(* IEC 61131-3 sources: uPC2_EMCTEST/UPC2_EMCTEST/UPC2_EMCTEST/Source/Programs, 11 files *)

(* ---- HeosTestMain.st ---- *)
USING System.UI;
USING System.IO;
USING System.EVD;
USING Libs.AinMng_v1_0_14;
USING libs.EVD_EVO_PosVlvs;

(* USING System.GwWifi; *)
USING System.RemoteIO;
USING System.Net.Plan;
USING System.Timer;
USING System.Text;
USING System;
USING System.Math;
USING System.PowerManagement;
USING System.Encoding;
USING System.NVRAM;
USING System.FileSystem;
USING System.FileSystem.Enums;

(* Constant defines *)
{DEFINE VALVE_NUM  2}
{DEFINE VALVE_MAX_VAL 1000}
{DEFINE VALVE_STATUS_INIT 0}
{DEFINE VALVE_STATUS_ZEROING 1}
{DEFINE VALVE_STATUS_OPER 2}
{DEFINE VALVE_STATUS_TEST_FAST_OPEN 3}
{DEFINE VALVE_STATUS_TEST_FAST_CLOSE 4}

//{DEFINE U_INPUT_NUM  12}
{DEFINE U_INPUT_NUM  16}
{DEFINE A_OUT_NUM  5}
{DEFINE D_OUT_NUM  13}
{DEFINE D_IN_NUM  10}

{DEFINE OUT_0_10V_HMI 254}

{DEFINE TEST_TIME_TIME 1000 }

TYPE
    (** I/O config *)
	InputConfigT : STRUCT
		IType : USINT;
        Mode : USINT;
        Filter : USINT;
		IMax,Imin : real;
	END_STRUCT;
END_TYPE

VAR_GLOBAL RETAIN
   SystemInited : BOOL;
   InputConfig : ARRAY[1..U_INPUT_NUM] OF InputConfigT;
   DOutStatus : ARRAY[1..D_OUT_NUM] OF BOOL:=[TRUE,TRUE,TRUE,TRUE,TRUE,TRUE,TRUE,TRUE,TRUE,TRUE,TRUE,TRUE,TRUE];
   AOutValue : ARRAY[1..A_OUT_NUM] OF REAL :=[5.0,6.0,8.0,5.0,6.0];
   UniAOutValue : ARRAY[1..U_INPUT_NUM] OF INT (0..1000);
   EvdAutoSwing : bool;
   EvdAutoSwingRandom : bool;
   { METADATA MAX_VAL 7}
   { METADATA MIN_VAL 0}
   RGB_LedStatus : INT; /* b2=R, b1=G, b0=B */
   GatewayOnOff : BOOL;
   Enable7SegLedToggle : bool;
   SegLedStat : bool;
   { METADATA MAX_VAL 500}
   { METADATA MIN_VAL 1}
   EvdAutoSwingSteps : INT;
   EnableTestTimer : bool := FALSE;
END_VAR

VAR_GLOBAL RETAIN
 RetainTestBuffer1 : ARRAY[1..1000] OF BYTE;
 RetainTestMaxIdx : uint:=0;
END_VAR

VAR_GLOBAL
 FirstCycle : bool := TRUE;
 EvdAutoSwingFast : bool:=TRUE;
 Cpcoe1_Err,Cpcoe2_Err,Cpcoe3_Err,Display_Err,BMS1_Err,ETH1_Err : BOOL;
 cPCOe1_ErrCode, cPCOe2_ErrCode, cPCOe3_ErrCode : INT;
 cPCOe1_CH1Val, cPCOe2_CH1Val, cPCOe3_CH1Val : REAL;
 InputValueI : ARRAY [1..U_INPUT_NUM] OF INT;
 InputValueR : ARRAY [1..U_INPUT_NUM] OF REAL;
 DInputValue : ARRAY [1..D_IN_NUM] OF BOOL;
 DefaultDInputValue : ARRAY [1..D_IN_NUM] OF BOOL := [FALSE, TRUE, FALSE, TRUE, FALSE, FALSE, FALSE, TRUE, FALSE, TRUE];

 Evd_struct: ARRAY [1..VALVE_NUM] OF TEEV;
 Evd_status : ARRAY [1..VALVE_NUM] OF USINT;
 Evd_instance : UNIPVLV_DRV;
 Evd_last_exec : ARRAY [1..VALVE_NUM] OF UDINT;
 Evd_Alm:ARRAY [1..2] OF BOOL;

 EVD_EVO_DevCfg : Libs.EVD_EVO_PosVlvs_v1_0_2.CFG_EVD;
 EVD_EVO_TypEEV : libs.EVD_EVO_PosVlvs_v1_0_2.EXV_VALVE:=libs.EVD_EVO_PosVlvs_v1_0_2.EXV_VALVE#CAREL_EXV;
 { METADATA MAX_VAL 1000}
 { METADATA MIN_VAL 0}
 EVD_EVO_PositionA_Msk : UINT;
 { METADATA MAX_VAL 1000}
 { METADATA MIN_VAL 0}
 EVD_EVO_PositionB_Msk : UINT;
 EVD_EVO_AutoSwingFast : BOOL:=TRUE;
 EVD_EVO_S1Value, EVD_EVO_S2Value, EVD_EVO_S3Value, EVD_EVO_S4Value : REAL;
 EVD_EVO_PositionA, EVD_EVO_PositionB, EVD_EVO_CurPositionA, EVD_EVO_CurPositionB, EVD_EVO_AutoStatusA, EVD_EVO_AutoStatusB: UINT;
 EVD_EVO_VarPositionB, EVD_EVO_VarPositionA,EVD_EVO_DevErr : INT;
 EVD_EVO_EEVParams : libs.EVD_Emb_Basic_v1_0_0.TEEV_PARAMS;
 EVD_EVO_Alr : libs.EVD_EVO_PosVlvs_v1_0_2.EVD_ALR;
 EVD_EVO_MBSErr : Libs.EVD_EVO_PosVlvs_v1_0_2.ModbusErrors;
 EVD_EVO_IO : Libs.EVD_EVO_PosVlvs_v1_0_2.EVD_IO;
 EVD_EVO_Ready,EVD_EVO_Online, EVD_EVO_Offline, EVD_EVO_ExV_Carel,EVD_EVO_SingleTwin,EVD_EVO_isEvdTwin,EVD_EVO_MstOffVlvClosed,EVD_EVO_S1Alarm,EVD_EVO_S2Alarm,EVD_EVO_S3Alarm,EVD_EVO_S4Alarm : BOOL;

 Evd_position : ARRAY [1..VALVE_NUM] OF INT (0..1000);
 AinAlarms:ARRAY [0..40] OF BOOL;
 EVD_EVOinstance : EvdEvo_PosVlvs;

 InputValAlarms:ARRAY [0..40] OF BOOL;
 { METADATA MAX_VAL 1000}
 { METADATA MIN_VAL 0}

 CurrentIOInfo: fwinfo;
 MyUUID : LWORD;
 MyUUID_H : DWORD;
 MyUUID_L : DWORD;
 MyUUID_STR : ARRAY[1..16] OF BYTE;
 MyUUID_S :  STRING;
 CurrentChipIoErrorInfo : ChipIoErrorInfo;
 ChipIoErrorCfg : ARRAY [1..5] OF UDINT(0..999);
 ChipIoErrorCrc : ARRAY [1..5] OF UDINT(0..999);
 ChipIoErrorNoasw : ARRAY [1..5] OF UDINT(0..999);
 ChipIoErrorExcep : ARRAY [1..5] OF UDINT(0..999);
 ChipIoErrorConsec : ARRAY [1..5] OF UDINT(0..999);
 ChipIoErrorCfgNolim : ARRAY [1..5] OF UDINT;
 ChipIoErrorCrcNolim : ARRAY [1..5] OF UDINT;
 ChipIoErrorNoaswNolim : ARRAY [1..5] OF UDINT;
 ChipIoErrorExcepNolim : ARRAY [1..5] OF UDINT;
 ChipIoErrorConsecNolim : ARRAY [1..5] OF UDINT;

 TotalChipIoError : uint;

 ErrorInfoLen : int;

 Ctime : DATE_AND_TIME;
 LYear, LMonth, LDay, LHour, LMin, LSec, LMs : UINT;
 WorkingTime :  UDINT;
 { METADATA MAX_VAL 60}
 { METADATA MIN_VAL 0}
 WorkingTimeSec : UINT;
 WorkingTimeMin : UINT;
 ToggleTime : UDINT;
 Toggle : bool;

// HeosSlaveSim_1: HeosSlaveSim;
 (*InverterCpu_01 : InverterCpu;
 InverterSecur_02 : InverterSecur;     *)
 Cpcoe_1, Cpcoe_2, Cpcoe_3 : Cpcoe;
 ValveProbe : VavleDriver_probe;
// InvMotor_01 : MBM_TMPL_PWRP_uMOTOR;
// InvSafe_02 : MBM_TMPL_PWRP_uSAFE;

 pCOE_input_1 : INT;
 ComStatusFb1Slave : BOOL;
 ComErrorFb1Slave : UINT;
 ComStatusFb2Inverter1 : BOOL;
 ComErrorFb2Inverter1 : UINT;
 ComStatusFb2Inverter2 : BOOL;
 ComErrorFb2Inverter2 : UINT;
 DisplayIsOnline : bool;

 EvdAutoSwingValue : INT;

 EvdAutoSwingUp : BOOL;
 EvdSwingTimer : UDINT;

 VersionStr : STRING;

 PowerSupplyState : UINT;
 { METADATA MAX_VAL 999}
 { METADATA MIN_VAL 0}
 PowerSupplyFrequency : UINT;

// deviceType:UINT;(* device model *)
// boardType:UINT;(* board type *)
// machineType:UINT; (* Target machine type *)
// hwCode:UINT;   (* Target hardware code *)

HwInfo : HardwareDescription;
OemInfoD : OemInfo;
OemID_String1: STRING;
OemID_String2: STRING;
OVOemID_String1: STRING;
OVOemID_String2: STRING;

Infos:  ProductInfo;

RetainBusErrorCount : uint;
RetainWrIndex : uint;
RetainTestEnableWr : bool;
RetainTestEnableWrPrev : bool;
RetainTestEnableRd : bool;
RetainWrErrorCount : uint;

NVRAMTestEnable : bool;
NVRAMTestCurrIdx : udint;
NVVRAMErrorCount : uint;
NVRAMError : DINT;
NV_Data:BYTE ;
NV_ValueChange : usint;

NAND_FileTestEnable : bool;
NAND_FileTestStatus : usint :=0;
Nand_FileBaseName: STRING:='EmcTestFile';
Nand_FileName : STRING;
NandFileID : DINT;
NandFileWrSize : DINT;
NandFileBuffer:ARRAY [1..5000] OF BYTE;
NandFileErrorCount : uint;
NandFileCnfErrorCount : uint;
NandFileOpenErrorCount : uint;
NandFileWriteErrorCount : uint;
NandFileIndex : int;

TestTimer : UDINT;
TestTimerFirstCycle : bool := TRUE;
RetainIsBusy : bool;
END_VAR

VAR_GLOBAL
IR_113_DCBusVoltage : int;
END_VAR

TYPE DisplayStatus:
(
    SEARCH_SEV_SEGMENTS,
    SEARCH_PLAN,
    SEV_SEGMENTS,
    PLAN
);
END_TYPE
VAR_GLOBAL
    mDisplayInfo : Remote_HMIInfo;
    termConfig : UDINT;
    sevSegTon : TON;
    pgd1Ton : TON;
    commissioningToolConnected : BOOL;
    status : DisplayStatus := DisplayStatus#SEARCH_PLAN;
    BothTermOffline : TON;
END_VAR

(* Default values *)
FUNCTION LoadDefault : BOOL
    VAR_INPUT Restore : BOOL;
    END_VAR
    VAR
        i : INT;
    END_VAR
    IF NOT SystemInited THEN
        SystemInited := TRUE;
    (* custom init for EMC test setup *)
    FOR i:=1 TO U_INPUT_NUM  DO

        CASE i OF
         1,2,4,5,7,10,11,12,14,15,16:
            InputConfig[i].IType := LIB_IO_PROBE_NTC;
         3,13:
            InputConfig[i].IType := LIB_IO_PROBE_0_5V;
            InputConfig[i].IMax := 5.0;
            InputConfig[i].Imin:=  0.0;
         8:
            InputConfig[i].IType := LIB_IO_PROBE_0_10V;
            InputConfig[i].IMax := 10.0;
            InputConfig[i].Imin:=  0.0;
         6:
            InputConfig[i].IType := LIB_IO_PROBE_0_1V;
            InputConfig[i].IMax := 1.0;
            InputConfig[i].Imin:=  0.0;
         9:
            InputConfig[i].IType := LIB_IO_PROBE_4_20MA;
            InputConfig[i].IMax := 20.0;
            InputConfig[i].Imin:=  4.0;
        END_CASE;
        (*InputConfig[i].IType := LIB_IO_PROBE_NTC;*)
        InputConfig[i].Mode := LIB_IO_AIN;
        InputConfig[i].Filter := 5;
//        InputConfig[i].IMax := 100.0;
//        InputConfig[i].Imin:=  0.0;

    END_FOR;
    END_IF;
EvdAutoSwingSteps := 1;
LoadDefault:=TRUE;
END_FUNCTION

(* Manages pGD1 <> 7 seg switch: return true if at least one display is alive *)
(**
 *
 *
 *                                                       -------------------
 *                              ----------------------->|      Search 7     |<------------------------<------
 *                             |              ----------|      segments     |---------               |       |
 *                             |             |           -------------------          |              |       |
 *                             |             |                                        |              |       |
 *                             |             |                                        |              |       |
 *                          NO |         YES |                                        | NO           | NO    |
 *                             |             |                                        |              |       |
 *                             |             |                                        |              |       |
 *                             |            \|/                                      \|/             |       |
 *                             |    -------------------                      -------------------     |       | NO
 *                              ---|         7         |                 ---|      Search       |---         |
 *                                 |      segments     |                |   |       pLan        |            |
 *                                  -------------------                 |    -------------------             |
 *                                                                      |                                    |
 *                                                                  YES |                                    |
 *                                                                      |                                    |
 *                                                                      |                                    |
 *                                                                     \|/                                   |
 *                                                             -------------------                           |
 *                                                            |        pLan       |-------------------------
 *                                                            |                   |
 *                                                             -------------------
 *
 *
*)

FUNCTION DisplayAutoSwitch : BOOL

   /* Check if there is a commissioning tool connected on serial display */
    IF IsCommissioningToolPresent() = TRUE AND GetConnectionChannel() = TO_DINT(Serial.Serial_Channel#Serial0) THEN
        commissioningToolConnected := TRUE;
    ELSE
        commissioningToolConnected := FALSE;
    END_IF;

    CASE status OF
        DisplayStatus#SEARCH_SEV_SEGMENTS:
            Display.Start();
            GetDisplayInfo(mDisplayInfo);
            sevSegTon(IN := mDisplayInfo.Alive = FALSE AND commissioningToolConnected = FALSE, PT := t#5s);
            IF sevSegTon.Q THEN
                Display.Stop();
                status := DisplayStatus#SEARCH_PLAN;
                sevSegTon(IN := FALSE);
            ELSIF mDisplayInfo.Alive = TRUE OR commissioningToolConnected = TRUE THEN
                status := DisplayStatus#SEV_SEGMENTS;
                sevSegTon(IN := FALSE);
            END_IF;

        DisplayStatus#SEARCH_PLAN:
            termConfig := GetNetTerminalConfiguration();
            pgd1Ton(IN := termConfig = 0, PT := t#10s);
            IF pgd1Ton.Q THEN
                status := DisplayStatus#SEARCH_SEV_SEGMENTS;
                pgd1Ton(IN := FALSE);
            ELSIF termConfig > 0 THEN
                status := DisplayStatus#PLAN;
                pgd1Ton(IN := FALSE);
            END_IF;
        DisplayStatus#SEV_SEGMENTS:
            GetDisplayInfo(mDisplayInfo);
            IF mDisplayInfo.Alive = FALSE AND commissioningToolConnected = FALSE THEN
                status := DisplayStatus#SEARCH_SEV_SEGMENTS;
            END_IF;
        DisplayStatus#PLAN:
            termConfig := GetNetTerminalConfiguration();
            IF termConfig = 0 THEN
                status := DisplayStatus#SEARCH_SEV_SEGMENTS;
            END_IF;
    END_CASE;

(* return true if at least one display is on-line *)
DisplayAutoSwitch := mDisplayInfo.Alive OR (termConfig > 0);
END_FUNCTION

(************************************************************)
PROGRAM uPC2EMCMain
	(* Insert strategy here *)
VAR
    i : INT;
    tmpval : UDINT;
    Ain_Mng_1 :AinMng;

END_VAR;

   Display.Init(FALSE);
   Display.Read();
   Display.Write();

  (*++++++++++++++++++++++++++++++++++++++++++++++++++++++++++++++++++++++++++++++++++++++ *)
  (* First Cycle *)
  IF FirstCycle THEN
     FirstCycle := FALSE;
     SetPlanAddress(1);

     IOGetFwInfo (CurrentIOInfo);
     LoadDefault(FALSE);

     (* convert version information *)
     CurrentIOInfo.chip[1].fw := CurrentIOInfo.chip[1].fw MOD 256 + (CurrentIOInfo.chip[1].fw / 256)*100;
     CurrentIOInfo.chip[2].fw := CurrentIOInfo.chip[2].fw MOD 256 + (CurrentIOInfo.chip[2].fw / 256)*100;
     CurrentIOInfo.chip[3].fw := CurrentIOInfo.chip[3].fw MOD 256 + (CurrentIOInfo.chip[3].fw / 256)*100;
     CurrentIOInfo.chip[4].fw := CurrentIOInfo.chip[4].fw MOD 256 + (CurrentIOInfo.chip[4].fw / 256)*100;
     CurrentIOInfo.chip[5].fw := CurrentIOInfo.chip[5].fw MOD 256 + (CurrentIOInfo.chip[5].fw / 256)*100;

     MyUUID := ulint_to_LWORD(GetUniqueId());
     MyUUID_H := lword_to_DWORD(SHR(MyUUID,32));
     MyUUID_L := lword_to_DWORD(MyUUID);
     System.Encoding.HEX_TO_STRING(MyUUID_STR, 1, 8, MyUUID_H);
     System.Encoding.HEX_TO_STRING(MyUUID_STR, 9, 8, MyUUID_L);
     FOR i:=1 TO 16 DO
      MyUUID_S := MyUUID_S + char_to_string(BYTE_TO_CHAR(MyUUID_STR[i]));
     END_FOR;

  (* Remove  just for test*)
  (*IOGetFwInfo (CurrentIOInfo);*)
  GetHardwareDescription(HwInfo);

  (* Get and convert OEM Infos *)
  System.GetOemInfo(OemInfoD);
  OemID_String1 := '';
  OemID_String2 := '';
  FOR i:=4 TO 1 BY -1 DO
      OemID_String1 := OemID_String1 + char_to_string(HEX_TO_STRING(shr(OemInfoD.OemID[i],4))) + char_to_string(HEX_TO_STRING( OemInfoD.OemID[i] & BYTE#15));
  END_FOR;
  FOR i:=6 TO 5 BY-1 DO
      OemID_String1 := OemID_String1 + char_to_string(HEX_TO_STRING(shr(OemInfoD.OemID[i],4))) + char_to_string(HEX_TO_STRING( OemInfoD.OemID[i] & BYTE#15));
  END_FOR;
  FOR i:=8 TO 7 BY-1 DO
      OemID_String1 := OemID_String1 + char_to_string(HEX_TO_STRING(shr(OemInfoD.OemID[i],4))) + char_to_string(HEX_TO_STRING( OemInfoD.OemID[i] & BYTE#15));
  END_FOR;

  FOR i:=dint_to_int(UPPER_BOUND(OemInfoD.OemID,1)/2+1) TO dint_to_int(UPPER_BOUND(OemInfoD.OemID,1)) DO
      OemID_String2 := OemID_String2 + char_to_string(HEX_TO_STRING(shr(OemInfoD.OemID[i],4))) + char_to_string(HEX_TO_STRING( OemInfoD.OemID[i] & BYTE#15));
  END_FOR;

  OVOemID_String1 := '';
  OVOemID_String2 := '';
  FOR i:=4 TO 1 BY -1 DO
      OVOemID_String1 := OVOemID_String1 + char_to_string(HEX_TO_STRING(shr(OemInfoD.OV_OemID[i],4))) + char_to_string(HEX_TO_STRING( OemInfoD.OV_OemID[i] & BYTE#15));
  END_FOR;

  FOR i:=6 TO 5 BY -1 DO
      OVOemID_String1 := OVOemID_String1 + char_to_string(HEX_TO_STRING(shr(OemInfoD.OV_OemID[i],4))) + char_to_string(HEX_TO_STRING( OemInfoD.OV_OemID[i] & BYTE#15));
  END_FOR;
  FOR i:=8 TO 7 BY -1 DO
      OVOemID_String1 := OVOemID_String1 + char_to_string(HEX_TO_STRING(shr(OemInfoD.OV_OemID[i],4))) + char_to_string(HEX_TO_STRING( OemInfoD.OV_OemID[i] & BYTE#15));
  END_FOR;

  FOR i:=dint_to_int(UPPER_BOUND(OemInfoD.OV_OemID,1)/2+1) TO dint_to_int(UPPER_BOUND(OemInfoD.OV_OemID,1)) DO
      OVOemID_String2 := OVOemID_String2 + char_to_string(HEX_TO_STRING(shr(OemInfoD.OV_OemID[i],4))) + char_to_string(HEX_TO_STRING( OemInfoD.OV_OemID[i] & BYTE#15));
  END_FOR;

     (** I/O configure: copy HMI values to configuration structures *)
     (** Univesal I/O **)
     FOR i:=1 TO TO_INT(CurrentIOInfo.U)  DO
         IF(InputConfig[i].IType <> OUT_0_10V_HMI) THEN
           uConfig[i].mode_type:=InputConfig[i].IType;
           uConfig[i].mode_sel := InputConfig[i].Mode;
           uConfig[i].filter := InputConfig[i].Filter;
         ELSE
           (** Out 0-10V **)
           uConfig[i].mode_sel := LIB_IO_AOUT;
           uConfig[i].mode_type := LIB_IO_OUT_0_10V;
         END_IF;

     END_FOR;
    (** Y output **)
     FOR i:=1 TO TO_INT(CurrentIOInfo.Y)  DO
       yConfig[i].mode_type:= LIB_IO_OUT_0_10V;
     END_FOR;

     VersionStr := CONCAT(TO_STRING(__PROJ_VER_MAJOR__), '.');
     VersionStr := CONCAT(VersionStr, TO_STRING(__PROJ_VER_MINOR__));

    (* get product code from Topological EEprom *)
    System.GetProductInfo(Infos);

   // System.SetNameSetting('HeosBox0');   removed

   //  PROVA := System.Net.TcpIp.GetIPHostname( );

      EVD_EVO_isEvdTwin := TRUE;
      EVD_EVO_MstOffVlvClosed := FALSE;
//      EVD_EVO_TypEEV := Libs.EVD_EVO_PosVlvs_v1_0_2.EXV_VALVE#CAREL_EXV;
//      EVD_EVO_IO.RelayA_Command := TRUE;
//      EVD_EVO_IO.RelayB_Command := TRUE;

  END_IF; (* First cycle *)

 (*++++++++++++++++++++++++++++++++++++++++++++++++++++++++++++++++++++++++++++++++++++++ *)
 (* Display Autoswitch pgd1 / LED *)
  DisplayIsOnline:=DisplayAutoSwitch();

 (* toogles a variable just to make led in 7Seg display blinking*)
 IF( System.GetSystemTime() - ToggleTime > 1000 ) THEN
    ToggleTime:=System.GetSystemTime();

     IF Enable7SegLedToggle THEN
       Toggle :=NOT(Toggle);
     END_IF;

 END_IF;

 (*++++++++++++++++++++++++++++++++++++++++++++++++++++++++++++++++++++++++++++++++++++++ *)
 (* U input configure and read to int*)
  FOR i:=1 TO TO_INT(CurrentIOInfo.U)  DO
      IF( InputConfig[i].IType <> OUT_0_10V_HMI ) THEN

       //IF(uConfig[i].mode_type<>InputConfig[i].IType) THEN
        uConfig[i].mode_type := InputConfig[i].IType;
        uConfig[i].mode_sel  := LIB_IO_AIN;
       //END_IF;

        Ain_Mng_1(
            Ain       := U[i].r,
            AinType   := InputConfig[i].IType,
            PrbOffset := 0.0,
            MinVal:=InputConfig[i].Imin,
            MaxVal:=InputConfig[i].Imax,
            En_Ain    := TRUE,
            PrbVal    => InputValueR[i],
            PrbAlrm   => AinAlarms[i]
        );
      ELSE
       uConfig[i].mode_type := LIB_IO_OUT_0_10V;
       uConfig[i].mode_sel  := LIB_IO_AOUT;
       Uout[i] := int_to_uint(UniAOutValue[i]);
      END_IF;
  END_FOR;

 (*++++++++++++++++++++++++++++++++++++++++++++++++++++++++++++++++++++++++++++++++++++++ *)
 (* Dig Out*)
 (* When EnableTestTimer is true NO 1 is used as timer measure output *)
  IF NOT EnableTestTimer  THEN
   FOR i:=1 TO TO_INT(CurrentIOInfo.NO) DO
        NO[i] := DOutStatus[i];
   END_FOR;
  END_IF;

 (*++++++++++++++++++++++++++++++++++++++++++++++++++++++++++++++++++++++++++++++++++++++ *)
 (* Dig input*)
  FOR i:=1 TO TO_INT(CurrentIOInfo.ID) DO
      DInputValue[i] := ID[i];
  END_FOR;
  IF EVD_EVOinstance.DeviceEvdEvo.Info.isOnline THEN
      DInputValue[5] :=NOT EVD_EVO_IO.DI1_Status;
      DInputValue[6] :=NOT EVD_EVO_IO.DI2_Status;
  END_IF;

 (*++++++++++++++++++++++++++++++++++++++++++++++++++++++++++++++++++++++++++++++++++++++ *)
 (* Analog out input*)
  FOR i:=1 TO TO_INT(CurrentIOInfo.Y)  DO
    Y[i] :=TO_UINT(AOutValue[i]*100.0);
  END_FOR;

 (*++++++++++++++++++++++++++++++++++++++++++++++++++++++++++++++++++++++++++++++++++++++ *)
 (* Serial port*)
//   Supervisor_BMS2.Init();
//   Supervisor_BMS2.Read();
   pCOWeb_BMS1.Init();
   pCOWeb_BMS1.Read();

   MS_LocalNet.Init();
   MS_LocalNet.Read();

//   InverterLine.Init();
//   InverterLine.Read();

   Supervisor_ETH1.Init();
   Supervisor_ETH1.Read();

    Line_cPCOe2.Init();
    Line_cPCOe2.Read();

    Line_cPCOe3.Init();
    Line_cPCOe3.Read();

(*Update variables here*)

 (*++++++++++++++++++++++++++++++++++++++++++++++++++++++++++++++++++++++++++++++++++++++ *)
 (* Valve init and update*)
   FOR i:=1 TO VALVE_NUM DO
    CASE Evd_status[i] OF
       VALVE_STATUS_INIT:
        Evd_status[i] := VALVE_STATUS_ZEROING;
        Evd_struct[i].Enable := 1;
        Evd_struct[i].PositionToSet := 0;
        Evd_struct[i].PositionToSet := 0;
        Evd_struct[i].CurrentEstimatedPosition := 0;
        Evd_struct[i].VariationToSet := -500;
        Evd_struct[i].ClosingSteps := 500;
        Evd_struct[i].MaxSteps := 480; (* or con 0x4000 per half steps *)
        Evd_struct[i].MinSteps := 0; (* not used *)
        Evd_struct[i].NominalCurrent := 350; (* not used *)
        Evd_struct[i].HoldingCurrent := 50;  (* not used *)
        Evd_struct[i].DutyCycle := 30;
        Evd_struct[i].ClosingXSteps := 1; (* not used *)
        Evd_struct[i].DutyCycleEnable := 1;
        Evd_struct[i].FastClosingSpeed := 150;
        Evd_struct[i].FastClosingSpeedEnable := 1;
        Evd_struct[i].OpeningXSteps := 1; (* not used *)
        Evd_struct[i].Speed := 50;
        Evd_last_exec[i]:=System.GetSystemTime();
       VALVE_STATUS_ZEROING:
        IF Evd_struct[i].CurrentEstimatedPosition  = 0  AND (System.GetSystemTime() - Evd_last_exec[i]) > 4000 THEN;
           Evd_status[i] := VALVE_STATUS_OPER;
        END_IF;

       VALVE_STATUS_OPER:
        IF EvdAutoSwingFast THEN
           Evd_status[i] := VALVE_STATUS_TEST_FAST_OPEN;
        END_IF;

         IF EvdAutoSwing THEN
           tmpval := INT_TO_UDINT(EvdAutoSwingValue);
           tmpval := (tmpval *  UINT_TO_UDINT(Evd_struct[i].MaxSteps)) / VALVE_MAX_VAL;
           Evd_struct[i].PositionToSet := UDINT_TO_UINT(tmpval);
         ELSE
          IF(Evd_position[i] >= VALVE_MAX_VAL) THEN
              Evd_position[i] := VALVE_MAX_VAL;
          END_IF;
        (*  IF(Evd_position[i] < 0) THEN
            Evd_position[i] := 0;
          END_IF;*)

          IF EvdAutoSwingRandom THEN
            (* add random +- 75 value to current position *)
            tmpval := INT_TO_UDINT(Evd_position[i] + real_to_int(150.0 * (System.Util.Random( ) - 0.5)) );
          ELSE
            tmpval := INT_TO_UDINT(Evd_position[i]);
          END_IF;

          tmpval := (tmpval *  UINT_TO_UDINT(Evd_struct[i].MaxSteps)) / VALVE_MAX_VAL;
          Evd_struct[i].PositionToSet := UDINT_TO_UINT(tmpval);

        END_IF;

      VALVE_STATUS_TEST_FAST_OPEN:
        IF Evd_struct[i].CurrentEstimatedPosition = Evd_struct[i].MaxSteps THEN
           Evd_struct[i].PositionToSet := 0;
           Evd_status[i] := VALVE_STATUS_TEST_FAST_CLOSE;
        ELSE
           Evd_struct[i].PositionToSet := Evd_struct[i].MaxSteps;
        END_IF;
        IF NOT( EvdAutoSwingFast) THEN
            Evd_status[i] := VALVE_STATUS_OPER;
        END_IF;

      VALVE_STATUS_TEST_FAST_CLOSE:
        IF Evd_struct[i].CurrentEstimatedPosition = 0 THEN
           Evd_struct[i].PositionToSet := Evd_struct[i].MaxSteps;
           Evd_status[i] := VALVE_STATUS_TEST_FAST_OPEN;
          ELSE
           Evd_struct[i].PositionToSet := 0;
        END_IF;
        IF NOT( EvdAutoSwingFast) THEN
            Evd_status[i] := VALVE_STATUS_OPER;
        END_IF;
       END_CASE;

     Evd_instance(ValveNum := INT_TO_BYTE(i), EEVIN := Evd_struct[i]);
  END_FOR;

  IF EvdAutoSwing THEN
   IF( System.GetSystemTime() - EvdSwingTimer > 2 ) THEN
      EvdSwingTimer:=System.GetSystemTime();

      IF EvdAutoSwingUp AND  EvdAutoSwingValue  < 1000  THEN
         EvdAutoSwingValue := EvdAutoSwingValue + (VALVE_MAX_VAL*EvdAutoSwingSteps)/(uint_to_int(Evd_struct[1].MaxSteps));
      END_IF;

      IF NOT(EvdAutoSwingUp) AND  EvdAutoSwingValue  >= 1  THEN
         EvdAutoSwingValue := EvdAutoSwingValue - (VALVE_MAX_VAL*EvdAutoSwingSteps)/(uint_to_int(Evd_struct[1].MaxSteps));
      END_IF;

      IF EvdAutoSwingValue >= 1000  THEN
          EvdAutoSwingUp := FALSE;
      END_IF;
      IF EvdAutoSwingValue <= 0  THEN
          EvdAutoSwingUp := TRUE;
      END_IF;
   END_IF;

 END_IF;

    EVD_EVO_PositionA := EVD_EVO_PositionA_Msk * 480 / 1000;
    EVD_EVO_PositionB := EVD_EVO_PositionB_Msk * 480 / 1000;

    IF EVD_EVO_AutoSwingFast AND EVD_EVO_Ready THEN
        IF EVD_EVO_AutoStatusA=0 THEN
            EVD_EVO_AutoStatusA := 1;
        END_IF;
        IF EVD_EVO_AutoStatusB=0 THEN
            EVD_EVO_AutoStatusB := 1;
        END_IF;
        EVD_EVO_PositionA_Msk := 0;
        EVD_EVO_PositionA_Msk := 0;
        IF EVD_EVO_AutoStatusA=1 THEN
            IF EVD_EVO_CurPositionA=480 THEN
                EVD_EVO_PositionA := 0;
                EVD_EVO_AutoStatusA := 2;
            ELSE
                EVD_EVO_PositionA := 480;
            END_IF;
        END_IF;
        IF EVD_EVO_AutoStatusA=2 THEN
            IF EVD_EVO_CurPositionA=0 THEN
                EVD_EVO_PositionA := 480;
                EVD_EVO_AutoStatusA := 1;
            ELSE
                EVD_EVO_PositionA := 0;
            END_IF;
        END_IF;
        IF EVD_EVO_AutoStatusB=1 THEN
            IF EVD_EVO_CurPositionB=480 THEN
                EVD_EVO_PositionB := 0;
                EVD_EVO_AutoStatusB := 2;
            ELSE
                EVD_EVO_PositionB := 480;
            END_IF;
        END_IF;
        IF EVD_EVO_AutoStatusB=2 THEN
            IF EVD_EVO_CurPositionB=0 THEN
                EVD_EVO_PositionB := 480;
                EVD_EVO_AutoStatusB := 1;
            ELSE
                EVD_EVO_PositionB := 0;
            END_IF;
        END_IF;
    ELSE
        EVD_EVO_AutoStatusA := 0;
        EVD_EVO_AutoStatusB := 0;
    END_IF;

    EVD_EVOinstance(
        DevAddr_EVD                     := 198,
        DevCfg_EVD                      := EVD_EVO_DevCfg,
        TypEEV                          := EVD_EVO_TypEEV,
        ValveA_PositionToSet            := EVD_EVO_PositionA,
        ValveB_PositionToSet            := EVD_EVO_PositionB,
        IsEvdTwin                       := EVD_EVO_isEvdTwin,
        MstOfflineVlvClosed             := EVD_EVO_MstOffVlvClosed,
        En_FB                           := TRUE,
        ReadyToWork                     => EVD_EVO_Ready,
        ValveA_CurrentEstimatedPosition => EVD_EVO_CurPositionA,
        ValveA_VariationToSet           => EVD_EVO_VarPositionA,
        ValveB_CurrentEstimatedPosition => EVD_EVO_CurPositionB,
        ValveB_VariationToSet           => EVD_EVO_VarPositionB,
        EEV_Params                      => EVD_EVO_EEVParams,
        Alr                             => EVD_EVO_Alr,
        Online_EVD                      => EVD_EVO_Online,
        OfflineAlrm_EVD                 => EVD_EVO_Offline,
        ModbusErr                       => EVD_EVO_MBSErr,
        ExV_Carel_Universal_Vlv         => EVD_EVO_ExV_Carel,
        EVD_Single_Twin                 => EVD_EVO_SingleTwin,
        IO                              := EVD_EVO_IO
    );
    EVD_EVO_DevErr :=TO_INT(EVD_EVOinstance.DeviceEvdEvo.Info.DeviceError);
    ValveProbe.Vlv_Probe_S1_ALARM_ENABLE := TRUE;
    ValveProbe.Vlv_Probe_S2_ALARM_ENABLE := TRUE;
    ValveProbe.Vlv_Probe_S3_ALARM_ENABLE := TRUE;
    ValveProbe.Vlv_Probe_S4_ALARM_ENABLE := TRUE;
    ValveProbe.Vlv_Probe_S1_ALARM_DELAY := 10;
    ValveProbe.Vlv_Probe_S2_ALARM_DELAY := 10;
    ValveProbe.Vlv_Probe_S3_ALARM_DELAY := 10;
    ValveProbe.Vlv_Probe_S4_ALARM_DELAY := 10;
    ValveProbe.Vlv_Probe_S1_PROBE_TYPE := 1;
    ValveProbe.Vlv_Probe_S3_PROBE_TYPE := 1;
    ValveProbe.Vlv_Probe_S2_PROBE_TYPE := 4;
    ValveProbe.Vlv_Probe_S4_PROBE_TYPE := 4;
    ValveProbe.Vlv_Probe_S1_RANGE_MAX := 4.5;
    ValveProbe.Vlv_Probe_S1_RANGE_MIN := 0.5;
    ValveProbe.Vlv_Probe_S3_RANGE_MAX := 4.5;
    ValveProbe.Vlv_Probe_S3_RANGE_MIN := 0.5;
    ValveProbe.Vlv_Probe_S1_ALARM_THRESHOLD_HIGH := 5.3;
    ValveProbe.Vlv_Probe_S1_ALARM_THRESHOLD_LOW := 4.7;
    ValveProbe.Vlv_Probe_S2_ALARM_THRESHOLD_HIGH := 100;
    ValveProbe.Vlv_Probe_S2_ALARM_THRESHOLD_LOW := 0;
    ValveProbe.Vlv_Probe_S3_ALARM_THRESHOLD_HIGH := 5.3;
    ValveProbe.Vlv_Probe_S3_ALARM_THRESHOLD_LOW := 4.7;
    ValveProbe.Vlv_Probe_S4_ALARM_THRESHOLD_HIGH := 100;
    ValveProbe.Vlv_Probe_S4_ALARM_THRESHOLD_LOW := 0;
    EVD_EVO_S1Value := ValveProbe.Vlv_Probe_S1_VALUE;
    EVD_EVO_S2Value := ValveProbe.Vlv_Probe_S2_VALUE;
    EVD_EVO_S3Value := ValveProbe.Vlv_Probe_S3_VALUE;
    EVD_EVO_S4Value := ValveProbe.Vlv_Probe_S4_VALUE;
    EVD_EVO_S1Alarm := ValveProbe.Vlv_Probe_S1_ALARM;
    EVD_EVO_S2Alarm := ValveProbe.Vlv_Probe_S2_ALARM;
    EVD_EVO_S3Alarm := ValveProbe.Vlv_Probe_S3_ALARM;
    EVD_EVO_S4Alarm := ValveProbe.Vlv_Probe_S4_ALARM;
 (*++++++++++++++++++++++++++++++++++++++++++++++++++++++++++++++++++++++++++++++++++++++ *)
 (* Update clock variables *)

 System.timer.GetTime(Ctime);
 System.Timer.SPLIT_DT(Ctime, LYear, LMonth, LDay, LHour, LMin, LSec, LMs);
 WorkingTime:=System.GetSystemTime()/1000;
 WorkingTimeSec := UDINT_TO_UINT((WorkingTime) MOD 60);
 WorkingTimeMin := UDINT_TO_UINT((WorkingTime) / 60);

 (*++++++++++++++++++++++++++++++++++++++++++++++++++++++++++++++++++++++++++++++++++++++ *)
 (* Update chipIo error infos *)
 (* get chipIO cfg errors*)

 TotalChipIoError := 0;
 ErrorInfoLen:=IOGetChipIoErrorInfo(0,ChipIoErrorCfgNoLim);
 FOR i:=1 TO 5 DO
  ChipIoErrorCfg[i] := ChipIoErrorCfgNoLim[i];
  TotalChipIoError := TotalChipIoError + udint_to_uint(ChipIoErrorCfgNoLim[i]);
 END_FOR;
 (* get chipIO comm CRC  errors*)
 ErrorInfoLen:=IOGetChipIoErrorInfo(1,ChipIoErrorCrcNoLim);
 FOR i:=1 TO 5 DO
  ChipIoErrorCrc[i] := ChipIoErrorCrcNoLim[i];
  TotalChipIoError := TotalChipIoError + udint_to_uint(ChipIoErrorCrcNoLim[i]);
 END_FOR;
 (* get chipIO comm no answer  errors*)
 ErrorInfoLen := IOGetChipIoErrorInfo(2, ChipIoErrorNoaswNoLim);
  FOR i:=1 TO 5 DO
  ChipIoErrorNoasw[i] := ChipIoErrorNoaswNoLim[i];
  TotalChipIoError := TotalChipIoError + udint_to_uint(ChipIoErrorNoaswNoLim[i]);
 END_FOR;
 (* get chipIO comm exception  errors*)
 ErrorInfoLen := IOGetChipIoErrorInfo(3, ChipIoErrorExcepNoLim);
 FOR i:=1 TO 5 DO
  ChipIoErrorExcep[i] := ChipIoErrorExcepNoLim[i];
   TotalChipIoError := TotalChipIoError + udint_to_uint(ChipIoErrorExcepNoLim[i]);
 END_FOR;

// HeosSlaveSim_1.HoldingRegister_CH1_TYPE := 0;
// pCOE_input_1 := HeosSlaveSim_1.HoldingRegister_CH1_VALUE;
// ComStatusFb1Slave  := HeosSlaveSim_1.Info.IsOnline;
// ComErrorFb1Slave := HeosSlaveSim_1.Info.ErrorsCount;
    Cpcoe_1.UnivChs_ChTyp[1] := 0;
    Cpcoe_1.DOuts_VALUE[1] := 1;
    cPCOe1_CH1Val := Cpcoe_1.UnivChs_VALUE[1];
    Cpcoe_2.UnivChs_ChTyp[1] := 0;
    Cpcoe_2.DOuts_VALUE[1] := 1;
    cPCOe2_CH1Val := Cpcoe_2.UnivChs_VALUE[1];
    Cpcoe_3.UnivChs_ChTyp[1] := 0;
    Cpcoe_3.DOuts_VALUE[1] := 1;
    cPCOe3_CH1Val := Cpcoe_3.UnivChs_VALUE[1];

(*Update variables here*)
(*InverterCpu_01.HoldingRegister_0 := 0;
ComStatusFb2Inverter1:=InverterCpu_01.Info.IsOnline;
ComErrorFb2Inverter1 := InverterCpu_01.Info.ErrorsCount;*)

//ComStatusFb2Inverter1:=InvMotor_01.Info.IsOnline;
//ComErrorFb2Inverter1 := InvMotor_01.Info.ErrorsCount;
//ComStatusFb2Inverter2:=InvSafe_02.Info.IsOnline;
//ComErrorFb2Inverter2 := InvSafe_02.Info.ErrorsCount;

MS_LocalNet.Write();
//InverterLine.Write();
//Supervisor_BMS2.Write();
pCOWeb_BMS1.Write();
Supervisor_ETH1.Write();
Line_cPCOe2.Write();
Line_cPCOe3.Write();

cPCOe1_ErrCode :=TO_INT(Cpcoe_1.Info.DeviceError);
cPCOe2_ErrCode:=TO_INT(Cpcoe_2.Info.DeviceError);
cPCOe3_ErrCode:=TO_INT(Cpcoe_3.Info.DeviceError);
Cpcoe1_Err := NOT Cpcoe_1.Info.isOnline OR cPCOe1_ErrCode <> 0;
Cpcoe2_Err := NOT Cpcoe_2.Info.isOnline OR cPCOe2_ErrCode <> 0;
Cpcoe3_Err := NOT Cpcoe_3.Info.isOnline OR cPCOe3_ErrCode <> 0;
//Display_Err := NOT Display.Info.Online;
BMS1_Err := NOT pCOWeb_BMS1.Info.Online;
ETH1_Err := NOT Supervisor_ETH1.Info.Online;

CASE  PowerManagement.GetPowerSupplyState() OF
    PowerSupplyState#UNKNOWN_PS: PowerSupplyState := 0;
    PowerSupplyState#AC_PS: PowerSupplyState := 1;
    PowerSupplyState#DC_PS: PowerSupplyState := 2;
    PowerSupplyState#AC_FAIL_PS: PowerSupplyState := 3;
    PowerSupplyState#DC_FAIL_PS: PowerSupplyState := 4;
END_CASE;
PowerSupplyfrequency := usint_to_uint(PowerManagement.GetPowerSupplyFrequency());

/* RGB led control */
//RGB.SetRGBLed(0,  int_to_byte(RGB_LedStatus/4 MOD 2), int_to_byte(RGB_LedStatus/2 MOD 2), int_to_byte(RGB_LedStatus MOD 2));

/* Gateway ON/OFF */
IF NOT EnableTestTimer  THEN
 IF( GatewayOnOff = 1) THEN
  SetGatewayWifiStatus(1);
 ELSE
  SetGatewayWifiStatus(0);
 END_IF;
END_IF;

(*------------------------------------------------*)
(* Retrieve model information *)
GetModel(deviceType, boardType, machineType, hwCode);

(*------------------------------------------------*)
(* Gather retain EEprom error using custom Exception manager, frequent writings need to be activated *)
IF (RetainTestEnableWr) THEN

  (* When set enable a clear is forced *)
  IF NOT(RetainTestEnableWrPrev) THEN
    FOR i:=1 TO dint_to_int(UPPER_BOUND(RetainTestBuffer1,1)) DO
         RetainTestBuffer1[i] := 0;
    END_FOR;
    RetainForceBackup();
    RetainTestEnableWrPrev := TRUE;
  END_IF;

 (* if exceptionmanger detects an write error on RETAIN RetainBusErrorCount is incremented*)
 IF EEpRetainErrorOccurred THEN
   RetainBusErrorCount:=RetainBusErrorCount+1;
   EEpRetainErrorOccurred := FALSE;
 END_IF;

 RetainWrIndex := RetainWrIndex + 1;
 IF((RetainWrIndex < 1) OR (RetainWrIndex > dint_to_uint(UPPER_BOUND(RetainTestBuffer1,1))) )
  THEN
     RetainWrIndex := 1;
  END_IF;

 (* writes  Retain *)
 RetainTestBuffer1[RetainWrIndex] := uint_to_byte(RetainWrIndex);

 IF(RetainTestMaxIdx < RetainWrIndex)  THEN
   RetainTestMaxIdx:=RetainWrIndex;
 END_IF;

 RetainForceBackup();

ELSE
 RetainTestEnableWrPrev := FALSE;
END_IF; (* RetainTestEnable *)

(*
IF RetainTestEnableRd THEN
  RetainWrErrorCount := 0;
  IF RetainTestMaxIdx > dint_to_uint(UPPER_BOUND(RetainTestBuffer1,1)) THEN
    RetainTestMaxIdx := dint_to_uint(UPPER_BOUND(RetainTestBuffer1, 1));
  END_IF;
  FOR i:=1 TO uint_to_int(RetainTestMaxIdx) DO
   IF(RetainTestBuffer1[i] <> int_to_byte(i) ) THEN
       RetainWrErrorCount := RetainWrErrorCount + 1;
      END_IF;
  END_FOR;
END_IF;   RetainTestEnableRd *)

(*------------------------------------------------*)
(* Gather NVRAM / FRAM read/write errors *)
IF (NVRAMTestEnable) THEN
    IF NVRAMTestCurrIdx >= NVRAM_GetSize() THEN
       NVRAMTestCurrIdx := 0;
       NV_ValueChange := NV_ValueChange + 1;

    END_IF;

    NVRAMError:=NVRAM_WriteVar(NVRAMTestCurrIdx,udint_to_byte(NVRAMTestCurrIdx+usint_to_udint(NV_ValueChange)));
    IF NVRAMError <0 THEN
      NVVRAMErrorCount := NVVRAMErrorCount + 1;
    END_IF;
    NVRAMError:=NVRAM_ReadVar(NVRAMTestCurrIdx,NV_Data);
    IF NVRAMError <0 THEN
      NVVRAMErrorCount := NVVRAMErrorCount + 1;
    END_IF;
    IF(NV_Data <> (udint_to_byte(NVRAMTestCurrIdx+usint_to_udint(NV_ValueChange)))) THEN
      NVVRAMErrorCount := NVVRAMErrorCount + 1;
    END_IF;
    NVRAMTestCurrIdx := NVRAMTestCurrIdx + 1;
END_IF;

(*------------------------------------------------*)
(* Gather NAND read/write error *)
IF NAND_FileTestEnable  THEN

 CASE  NAND_FileTestStatus OF
    0: (* create and write *)
      NandFileIndex := NandFileIndex + 1;
       IF( NandFileIndex > 10) THEN
          NandFileIndex := 1;
       END_IF;
      Nand_FileName := Nand_FileBaseName + int_to_string(NandFileIndex) + '.bin';
      NandFileID:=FileOpen(PartitionType#PublicPartition,Nand_FileName,FS_OpenMode#CREATE_RW);
      IF NandFileID >= 0 THEN
         FOR i:=1 TO dint_to_int(UPPER_BOUND(NandFileBuffer,1)) DO
             NandFileBuffer[i]:=int_to_byte(i);
         END_FOR;
         NandFileWrSize:=FileWrite(NandFileID, NandFileBuffer);
         IF(NandFileWrSize <> 5000) THEN
             NandFileErrorCount := NandFileErrorCount + 1;
             NandFileWriteErrorCount := NandFileWriteErrorCount + 1;
         END_IF;
         FileClose(NandFileID);
      ELSE
        NandFileErrorCount := NandFileErrorCount + 1;
        NandFileOpenErrorCount := NandFileOpenErrorCount + 1;
      END_IF;
      NAND_FileTestStatus := 1;

    1: (* read and verify *)
      NandFileID:=FileOpen(PartitionType#PublicPartition,Nand_FileName,FS_OpenMode#OPEN_READ);
      IF NandFileID >= 0 THEN
        FOR i:=1 TO dint_to_int(UPPER_BOUND(NandFileBuffer,1)) DO
             NandFileBuffer[i]:=0;
        END_FOR;
        FileRead(NandFileID, NandFileBuffer);
        FOR i:=1 TO dint_to_int(UPPER_BOUND(NandFileBuffer,1)) DO
             IF( NandFileBuffer[i] <> int_to_byte(i)) THEN
                 NandFileErrorCount := NandFileErrorCount + 1;
                 NandFileCnfErrorCount := NandFileCnfErrorCount + 1;
                 EXIT;
             END_IF;
        END_FOR;
       FileClose(NandFileID);
      ELSE
        NandFileErrorCount := NandFileErrorCount + 1;
        NandFileOpenErrorCount := NandFileOpenErrorCount + 1;
      END_IF;
      NAND_FileTestStatus := 0;
END_CASE;

END_IF;

(* When EnableTestTimer is true NO 1 and GatewayWifiStatus are used as timer measure outputs *)
IF EnableTestTimer  THEN
  tmpval := GetSystemTime() - TestTimer;
  IF ( tmpval  >=  TEST_TIME_TIME ) THEN

   IF TestTimerFirstCycle THEN
       TestTimerFirstCycle := FALSE;
       tmpval := TEST_TIME_TIME;
   END_IF;
   TestTimer := GetSystemTime() - (tmpval  -  TEST_TIME_TIME);

   NO[1] := NOT NO[1];
   IF(NO[1]) THEN
      SetGatewayWifiStatus(1);
   ELSE
      SetGatewayWifiStatus(0);
   END_IF;
  END_IF;
 ELSE
  TestTimerFirstCycle := TRUE;
END_IF;

(* Refresh UI *)
SendVirtualKey(NO_KEY, 1);
END_PROGRAM

(* ---- 050_StoreAlarms.st ---- *)
USING System;
USING System.Math;
USING System.Alarm;
USING System.Timer;

USING Libs.Logics_v0_1_4;
USING Libs.Alarm_Mng_v1_1_5;

VAR_GLOBAL CONSTANT
    {REGION UPDATE EVERY TIME AN ALARM IS ADDEDD!}
        (**Number of alarm saved inside ALARM table.
         *NOTE: update every time an alarm is addedd!
        *)
        noAlrms : UINT := 50;
    {ENDREGION}

    {REGION ALARM LOG CONFIGURATION}
        (**Number of logs of alarms saved inside ALARM-LOG table*)
        noAlrmsLog     : UINT := 50;
        (**
         *Size of the array VARs_TO_LOG.
         *Number of additionals variables saved inside ALARM-LOG table,
         *when an alarm is triggered (NOTE: used inside System.Alarm library)
        *)
        MaxAlarmValues : UINT := 1;
    {ENDREGION}

    {REGION Alarm widget description}
        (**Alarm descriptions*)
        AlarmDescr : ARRAY[1..noAlrms] OF STRING[66] :=
                                                       (*  |-------Row 1---------|-------Row 2---------|-------Row 3--------| *)
                                                           [
                                                (*AL01*)   'System - RETAIN memory written too often.                         ',
                                                (*AL02*)   'System - NFC memory written too often.                            ',
                                                (*AL03*)   'U1-Probe Alarm                                                    ',
                                                (*AL04*)   'U2-Probe Alarm                                                    ',
                                                (*AL05*)   'U3-Probe Alarm                                                    ',
                                                (*AL06*)   'U4-Probe Alarm                                                    ',
                                                (*AL07*)   'U5-Probe Alarm                                                    ',
                                                (*AL08*)   'U6-Probe Alarm                                                    ',
                                                (*AL09*)   'U7-Probe Alarm                                                    ',
                                                (*AL10*)   'U8-Probe Alarm                                                    ',
                                                (*AL11*)   'U9-Probe Alarm                                                    ',
                                                (*AL12*)   'U10-Probe Alarm                                                   ',
                                                (*AL13*)   'DI1-Alarm                                                         ',
                                                (*AL14*)   'DI2-Alarm                                                         ',
                                                (*AL15*)   'DI3-Alarm                                                         ',
                                                (*AL16*)   'DI4-Alarm                                                         ',
                                                (*AL17*)   'DI5-Alarm                                                         ',
                                                (*AL18*)   'DI6-Alarm                                                         ',
                                                (*AL19*)   'DI7-Alarm                                                         ',
                                                (*AL20*)   'DI8-Alarm                                                         ',
                                                (*AL21*)   'DI9-Alarm                                                         ',
                                                (*AL22*)   'DI10-Alarm                                                        ',
                                                (*AL23*)   'U11-Probe Alarm                                                   ',
                                                (*AL24*)   'U12-Probe Alarm                                                   ',
                                                (*AL25*)   'U12-Probe Alarm                                                   ',
                                                (*AL26*)   'U12-Probe Alarm                                                   ',
                                                (*AL27*)   'cPCO1-Alarm                                                       ',
                                                (*AL28*)   'cPCO2-Alarm                                                       ',
                                                (*AL29*)   'cPCO3-Alarm                                                       ',
                                                (*AL30*)   'U1-Value Alarm                                                    ',
                                                (*AL31*)   'U2-Value Alarm                                                    ',
                                                (*AL32*)   'U3-Value Alarm                                                    ',
                                                (*AL33*)   'U4-Value Alarm                                                    ',
                                                (*AL34*)   'U5-Value Alarm                                                    ',
                                                (*AL35*)   'U6-Value Alarm                                                    ',
                                                (*AL36*)   'U7-Value Alarm                                                    ',
                                                (*AL37*)   'U8-Value Alarm                                                    ',
                                                (*AL38*)   'U9-Value Alarm                                                    ',
                                                (*AL39*)   'U10-Value Alarm                                                   ',
                                                (*AL40*)   'U11-Value Alarm                                                   ',
                                                (*AL41*)   'U12-Value Alarm                                                   ',
                                                (*AL42*)   'Display Connect Alarm                                             ',
                                                (*AL43*)   'BMS1 Connect Alarm                                                ',
                                                (*AL44*)   'ETH1 Connect Alarm                                                ',
                                                (*AL45*)   'Valve Driver Alarm                                                ',
                                                (*AL45*)   'S1 Alarm                                                          ',
                                                (*AL45*)   'S2 Alarm                                                          ',
                                                (*AL45*)   'S3 Alarm                                                          ',
                                                (*AL45*)   'S4 Alarm                                                          '
                                                           ];
        (**Stored variable 1 description*)
        StoreVarDesc1 : ARRAY[1..noAlrms] OF STRING[14]:=
                                                            [
                                                (*AL01*)    'Desc. Var1:',
                                                (*AL02*)    'Desc. Var1:',
                                                (*AL03*)    'Desc. Var1:',
                                                (*AL04*)    'Desc. Var1:'
                                                            ];
        (**Stored variable 2 description*) //StoreVarDesc2
        StoreVarDesc2 : ARRAY[1..noAlrms] OF STRING[14]:=
                                                            [
                                                (*AL01*)    'Desc. Var2:',
                                                (*AL02*)    'Desc. Var2:',
                                                (*AL03*)    'Desc. Var2:',
                                                (*AL04*)    'Desc. Var2:'
                                                            ];
    {ENDREGION}

    {REGION CONFIGURE HERE YOUR ALARMs CATEGORY (max 16). YOU NEED TO USE "ActAlr_ForCategory".}
        (**Alarm category associate to ActAlr_ForCategory BIT_0 *) CAT_FREE_0            : UINT := 1;
        (**Alarm category associate to ActAlr_ForCategory BIT_1 *) CAT_AL_SRS_UNIT       : UINT := 2;
        (**Alarm category associate to ActAlr_ForCategory BIT_2 *) CAT_AL_SRS_CIRC1      : UINT := 4;
        (**Alarm category associate to ActAlr_ForCategory BIT_3 *) CAT_PROBES            : UINT := 8;
        (**Alarm category associate to ActAlr_ForCategory BIT_4 *) CAT_WRG_REGUL         : UINT := 16;
        (**Alarm category associate to ActAlr_ForCategory BIT_5 *) CAT_WRG_BOARD_MST     : UINT := 32;
        (**Alarm category associate to ActAlr_ForCategory BIT_6 *) CAT_FREE_6            : UINT := 64;
        (**Alarm category associate to ActAlr_ForCategory BIT_7 *) CAT_WRG_CIRC1         : UINT := 128;
        (**Alarm category associate to ActAlr_ForCategory BIT_8 *) CAT_FREE_8            : UINT := 256;
        (**Alarm category associate to ActAlr_ForCategory BIT_9 *) CAT_FREE_9            : UINT := 512;
        (**Alarm category associate to ActAlr_ForCategory BIT_10*) CAT_WRG_HRSCOUNTER    : UINT := 1024;
        (**Alarm category associate to ActAlr_ForCategory BIT_11*) CAT_FREE_11           : UINT := 2048;
        (**Alarm category associate to ActAlr_ForCategory BIT_12*) CAT_FREE_12           : UINT := 4096;
        (**Alarm category associate to ActAlr_ForCategory BIT_13*) CAT_FREE_13           : UINT := 8192;
        (**Alarm category associate to ActAlr_ForCategory BIT_14*) CAT_FREE_14           : UINT := 16384;
        (**Alarm category associate to ActAlr_ForCategory BIT_15*) CAT_BLINK_KEY_SERVICE : UINT := 32768;
    {ENDREGION}
END_VAR

VAR_GLOBAL PERSISTENT
    (**Log alarm array*)
    Log_Alarm  : ARRAY[1..noAlrmsLog] OF AlarmLog;
    (**Index of Log_Alarm *)
    LogAlrmIdx : UINT;
END_VAR

VAR_GLOBAL
    {REGION ALARMS MANAGEMENT}
        (**Container of Alarms table*)
        Alarms              : AlarmUnion;
        (**Array of active alarms*)
        Active_Alrm         : ARRAY[1..noAlrms] OF UINT;
        (**Active alarm status for each category, max 16 differents category (Bit15..Bit0)*)
        ActAlr_ForCategory  : WORD;
    {ENDREGION}

    {REGION ALARM RESET}
        (**A request to reset all alarms is active (FALSE=NO, TRUE=Reset)*)
    	AlrmRes             : BOOL;
    	(**Reset active alarms by BMS net (FALSE=NO, TRUE=Reset)*)
    	ResAlrmByBMS        : BOOL;
    	(**Reset alarms by user interface (FALSE=NO, TRUE=Reset)*)
    	ResAlrmByHMI        : BOOL;
    {ENDREGION}

    {REGION ALARMS AND WARNINGS}
        {REGION ALARMS}
            (**RelayAlrm - Global alarm relay*)
        	RelayAlrm           : BOOL;
            (**Please call the SERVICE, a serius alarm is present inside the unit*)
        	Al_Call_Service     : BOOL;
        	(**Miscellaneous alarms*)
        	Al_MiscAlrms        : BOOL;
        	(**Regulation alarms*)
        	Al_RegulationAlrms  : BOOL;
        	(**Serious alarm circ.1*)
        	Al_SrsCirc1         : BOOL;
        	(**Unit serious alarm*)
        	Al_SrsUnit          : BOOL;
        {ENDREGION}

        {REGION WARNINGS}
            (**Warning - Master board alarm*)
        	Wrg_BoardMst    : BOOL;
        	(**Warning - Circ.1 light alarm*)
        	Wrg_Circ1       : BOOL;
        	(**Warning - Hours counters alarm is active*)
        	Wrg_HrsCounters : BOOL;
        	(**Warning - Regulation alarm*)
        	Wrg_Regul       : BOOL;
        {ENDREGION}
    {ENDREGION}

    {REGION ALARMS LOG}
        (**Array of variables to store inside LOG_ALARM array, when an alarm happen*)
        VARs_TO_LOG : ARRAY[0..MaxAlarmValues] OF AlarmValue;
        (**Empty structured used to clean LOG_ALARM array*)
        CleanLog    : AlarmLog;
        (**Alarms Log clear command (FALSE=No, TRUE=Yes)*)
    	LogAlrmRes  : BOOL;
    {ENDREGION}
END_VAR

VAR_GLOBAL INTERNAL
    (*Used by Modbus files transfer protocol*)
    AlrmInfoArr : ARRAY [1..noAlrms] OF AlarmInfo;
END_VAR

TYPE
    (**This structure manages all unit's alarms*)
    AlarmUnion : UNION
        (**Array of FBs Alarm_Req*)
        Arr   : ARRAY [1..noAlrms] OF Alarm_Req;
        (**Table of all alarms and them property*)
        Table : AlarmsStruct;
    END_UNION;

    (**List all alarms and them property (Code, Category, Reset type, ...)*)
    AlarmsStruct : STRUCT
            {REGION UNIT}
                (** A01 Unit - Retain memory saved too often*)
                Al_RetainSavedTooOften : Alarm_Req := (StrCode := 'A01', Info := (Code := 001, Category := CAT_AL_SRS_UNIT, Reset := AlarmResetType#Manual));
                (** A02 Unit - NFC memory saved too often*)
                Al_NFCSavedTooOften    : Alarm_Req := (StrCode := 'A02', Info := (Code := 002, Category := CAT_AL_SRS_UNIT, Reset := AlarmResetType#Manual));
                (** A03 Unit - Remote alarm by Din 1*)
                Al_U1_PrbAlrm            : Alarm_Req := (StrCode := 'A03', Info := (Code := 003, Category := CAT_PROBES, Reset := AlarmResetType#Auto));
                (** A04 Unit - Remote alarm by Din 1*)
                Al_U2_PrbAlrm            : Alarm_Req := (StrCode := 'A04', Info := (Code := 004, Category := CAT_PROBES, Reset := AlarmResetType#Auto));
                (** A05 Unit - Remote alarm by Din 1*)
                Al_U3_PrbAlrm            : Alarm_Req := (StrCode := 'A05', Info := (Code := 005, Category := CAT_PROBES, Reset := AlarmResetType#Auto));
                (** A06 Unit - Remote alarm by Din 1*)
                Al_U4_PrbAlrm            : Alarm_Req := (StrCode := 'A06', Info := (Code := 006, Category := CAT_PROBES, Reset := AlarmResetType#Auto));
                (** A07 Unit - Remote alarm by Din 1*)
                Al_U5_PrbAlrm            : Alarm_Req := (StrCode := 'A07', Info := (Code := 007, Category := CAT_PROBES, Reset := AlarmResetType#Auto));
                (** A08 Unit - Remote alarm by Din 1*)
                Al_U6_PrbAlrm            : Alarm_Req := (StrCode := 'A08', Info := (Code := 008, Category := CAT_PROBES, Reset := AlarmResetType#Auto));
                (** A09 Unit - Remote alarm by Din 1*)
                Al_U7_PrbAlrm            : Alarm_Req := (StrCode := 'A09', Info := (Code := 009, Category := CAT_PROBES, Reset := AlarmResetType#Auto));
                (** A10 Unit - Remote alarm by Din 1*)
                Al_U8_PrbAlrm            : Alarm_Req := (StrCode := 'A10', Info := (Code := 010, Category := CAT_PROBES, Reset := AlarmResetType#Auto));
                (** A11 Unit - Remote alarm by Din 1*)
                Al_U9_PrbAlrm            : Alarm_Req := (StrCode := 'A11', Info := (Code := 011, Category := CAT_PROBES, Reset := AlarmResetType#Auto));
                (** A12 Unit - Remote alarm by Din 1*)
                Al_U10_PrbAlrm            : Alarm_Req := (StrCode := 'A12', Info := (Code := 012, Category := CAT_PROBES, Reset := AlarmResetType#Auto));
                (** A13 Unit - Remote alarm by Din 1*)
                Al_DI1Alrm            : Alarm_Req := (StrCode := 'A13', Info := (Code := 013, Category := CAT_PROBES, Reset := AlarmResetType#Auto));
                (** A14 Unit - Remote alarm by Din 1*)
                Al_DI2Alrm            : Alarm_Req := (StrCode := 'A14', Info := (Code := 014, Category := CAT_PROBES, Reset := AlarmResetType#Auto));
                (** A15 Unit - Remote alarm by Din 1*)
                Al_DI3Alrm            : Alarm_Req := (StrCode := 'A15', Info := (Code := 015, Category := CAT_PROBES, Reset := AlarmResetType#Auto));
                (** A16 Unit - Remote alarm by Din 1*)
                Al_DI4Alrm            : Alarm_Req := (StrCode := 'A16', Info := (Code := 016, Category := CAT_PROBES, Reset := AlarmResetType#Auto));
                (** A17 Unit - Remote alarm by Din 1*)
                Al_DI5Alrm            : Alarm_Req := (StrCode := 'A17', Info := (Code := 017, Category := CAT_PROBES, Reset := AlarmResetType#Auto));
                (** A18 Unit - Remote alarm by Din 1*)
                Al_DI6Alrm            : Alarm_Req := (StrCode := 'A18', Info := (Code := 018, Category := CAT_PROBES, Reset := AlarmResetType#Auto));
                (** A19 Unit - Remote alarm by Din 1*)
                Al_DI7Alrm            : Alarm_Req := (StrCode := 'A19', Info := (Code := 019, Category := CAT_PROBES, Reset := AlarmResetType#Auto));
                (** A20 Unit - Remote alarm by Din 1*)
                Al_DI8Alrm            : Alarm_Req := (StrCode := 'A20', Info := (Code := 020, Category := CAT_PROBES, Reset := AlarmResetType#Auto));
                (** A21 Unit - Remote alarm by Din 1*)
                Al_DI9Alrm            : Alarm_Req := (StrCode := 'A21', Info := (Code := 021, Category := CAT_PROBES, Reset := AlarmResetType#Auto));
                (** A22 Unit - Remote alarm by Din 1*)
                Al_DI10Alrm            : Alarm_Req := (StrCode := 'A22', Info := (Code := 022, Category := CAT_PROBES, Reset := AlarmResetType#Auto));
                (** A23 Unit - Remote alarm by Din 1*)
                Al_U11_PrbAlrm            : Alarm_Req := (StrCode := 'A23', Info := (Code := 023, Category := CAT_PROBES, Reset := AlarmResetType#Auto));
                (** A24 Unit - Remote alarm by Din 1*)
                Al_U12_PrbAlrm            : Alarm_Req := (StrCode := 'A24', Info := (Code := 024, Category := CAT_PROBES, Reset := AlarmResetType#Auto));
                (** A25 Unit - Room temperature probe alarm by Ain 1*)
                Al_Ain1Alrm            : Alarm_Req := (StrCode := 'A25', Info := (Code := 025, Category := CAT_PROBES, Reset := AlarmResetType#Auto));
                (** A26 Unit - Room temperature probe alarm by Ain 1*)
                Al_HiTemp              : Alarm_Req := (StrCode := 'A26', Info := (Code := 026, Category := CAT_PROBES,   Reset := AlarmResetType#Auto));
                (** A27 Unit - Room temperature probe alarm by Ain 1*)
                Al_cPCOe1ERR            : Alarm_Req := (StrCode := 'A27', Info := (Code := 027, Category := CAT_AL_SRS_UNIT, Reset := AlarmResetType#Auto));
                (** A28 Unit - Room temperature probe alarm by Ain 1*)
                Al_cPCOe2ERR            : Alarm_Req := (StrCode := 'A28', Info := (Code := 028, Category := CAT_AL_SRS_UNIT, Reset := AlarmResetType#Auto));
                (** A28 Unit - Room temperature probe alarm by Ain 1*)
                Al_cPCOe3ERR            : Alarm_Req := (StrCode := 'A29', Info := (Code := 029, Category := CAT_AL_SRS_UNIT, Reset := AlarmResetType#Auto));
                (** A23 Unit - Remote alarm by Din 1*)
                Al_U1_ValAlrm            : Alarm_Req := (StrCode := 'A30', Info := (Code := 030, Category := CAT_PROBES, Reset := AlarmResetType#Auto));
                (** A24 Unit - Remote alarm by Din 1*)
                Al_U2_valAlrm            : Alarm_Req := (StrCode := 'A31', Info := (Code := 031, Category := CAT_PROBES, Reset := AlarmResetType#Auto));
                (** A23 Unit - Remote alarm by Din 1*)
                Al_U3_ValAlrm            : Alarm_Req := (StrCode := 'A32', Info := (Code := 032, Category := CAT_PROBES, Reset := AlarmResetType#Auto));
                (** A24 Unit - Remote alarm by Din 1*)
                Al_U4_ValAlrm            : Alarm_Req := (StrCode := 'A33', Info := (Code := 033, Category := CAT_PROBES, Reset := AlarmResetType#Auto));
                (** A23 Unit - Remote alarm by Din 1*)
                Al_U5_ValAlrm            : Alarm_Req := (StrCode := 'A34', Info := (Code := 034, Category := CAT_PROBES, Reset := AlarmResetType#Auto));
                (** A24 Unit - Remote alarm by Din 1*)
                Al_U6_ValAlrm            : Alarm_Req := (StrCode := 'A35', Info := (Code := 035, Category := CAT_PROBES, Reset := AlarmResetType#Auto));
                (** A23 Unit - Remote alarm by Din 1*)
                Al_U7_ValAlrm            : Alarm_Req := (StrCode := 'A36', Info := (Code := 036, Category := CAT_PROBES, Reset := AlarmResetType#Auto));
                (** A24 Unit - Remote alarm by Din 1*)
                Al_U8_ValAlrm            : Alarm_Req := (StrCode := 'A37', Info := (Code := 037, Category := CAT_PROBES, Reset := AlarmResetType#Auto));
                (** A23 Unit - Remote alarm by Din 1*)
                Al_U9_ValAlrm            : Alarm_Req := (StrCode := 'A38', Info := (Code := 038, Category := CAT_PROBES, Reset := AlarmResetType#Auto));
                (** A24 Unit - Remote alarm by Din 1*)
                Al_U10_ValAlrm            : Alarm_Req := (StrCode := 'A39', Info := (Code := 039, Category := CAT_PROBES, Reset := AlarmResetType#Auto));
                (** A23 Unit - Remote alarm by Din 1*)
                Al_U11_ValAlrm            : Alarm_Req := (StrCode := 'A40', Info := (Code := 040, Category := CAT_PROBES, Reset := AlarmResetType#Auto));
                (** A24 Unit - Remote alarm by Din 1*)
                Al_U12_ValAlrm            : Alarm_Req := (StrCode := 'A41', Info := (Code := 041, Category := CAT_PROBES, Reset := AlarmResetType#Auto));
                (** A27 Unit - Room temperature probe alarm by Ain 1*)
                Al_DisplayERR            : Alarm_Req := (StrCode := 'A42', Info := (Code := 042, Category := CAT_AL_SRS_UNIT, Reset := AlarmResetType#Auto));
                (** A27 Unit - Room temperature probe alarm by Ain 1*)
                Al_BMS1ERR            : Alarm_Req := (StrCode := 'A43', Info := (Code := 043, Category := CAT_AL_SRS_UNIT, Reset := AlarmResetType#Auto));
                (** A27 Unit - Room temperature probe alarm by Ain 1*)
                Al_ETH1ERR            : Alarm_Req := (StrCode := 'A44', Info := (Code := 044, Category := CAT_AL_SRS_UNIT, Reset := AlarmResetType#Auto));
                (** A27 Unit - Room temperature probe alarm by Ain 1*)
                Al_ValveDriveERR      : Alarm_Req := (StrCode := 'A45', Info := (Code := 045, Category := CAT_AL_SRS_UNIT, Reset := AlarmResetType#Auto));
                (** A24 Unit - Remote alarm by Din 1*)
                Al_S1_Alrm            : Alarm_Req := (StrCode := 'A46', Info := (Code := 046, Category := CAT_PROBES, Reset := AlarmResetType#Auto));
                (** A24 Unit - Remote alarm by Din 1*)
                Al_S2_Alrm            : Alarm_Req := (StrCode := 'A47', Info := (Code := 047, Category := CAT_PROBES, Reset := AlarmResetType#Auto));
                (** A24 Unit - Remote alarm by Din 1*)
                Al_S3_Alrm            : Alarm_Req := (StrCode := 'A48', Info := (Code := 048, Category := CAT_PROBES, Reset := AlarmResetType#Auto));
                (** A24 Unit - Remote alarm by Din 1*)
                Al_S4_Alrm            : Alarm_Req := (StrCode := 'A49', Info := (Code := 049, Category := CAT_PROBES, Reset := AlarmResetType#Auto));
            {ENDREGION}

            (** -----------------------
                ADD HERE YOUR ALARMS!
            ---------------------------*)
    END_STRUCT;
END_TYPE

(**This program manages alarm categories and detects the alarms*)
PROGRAM StoreAlarms
    VAR_TEMP
        (**Numeber of alarm active*)
        TotActAlm : UINT;
    END_VAR

    VAR
        (**Array index*)
        idx             : DINT;

        (**Numeber of alarm active in previous cycle*)
        TotActAlm_Old   : UINT;

        TP_ResAlrmByBMS : TP;

        {REGION USED BY LOG-ALARM TO STORE THE "ADDITIONAL VARIABLES"}
        (**A01 trigger used to store additional values*)
        RFtrg_Alr1       : RF_TRIG;
        (**A02 trigger used to store additional values*)
        RFtrg_Alr2       : RF_TRIG;
        (**A03 trigger used to store additional values*)
        RFtrg_Alr3       : RF_TRIG;
        (**A04 trigger used to store additional values*)
        RFtrg_Alr4       : RF_TRIG;
        {ENDREGION}
    END_VAR

    {REGION RESET ALARM ARRAY}
        TP_ResAlrmByBMS(IN := ResAlrmByBMS, PT := T#5s);        (*Request of reset by BMS*)
        ResAlrmByBMS := TP_ResAlrmByBMS.Q;

        AlrmRes := ResAlrmByBMS OR ResAlrmByHMI;
    {ENDREGION}

    {REGION GET ACTIVE ALARMS}
        FOR idx := 1 TO UPPER_BOUND(Alarms.Arr, 1) DO
            {REGION IoT Third Parts Integration: Alarms retrieve via "Modbus File Transfer"}
                AlrmInfoArr[idx] := Alarms.Arr[idx].Info;       (*Copy the alarm info into a dedicated array*)
            {ENDREGION}

            {REGION "ADDITIONAL VARIABLES" stored inside LOG_ALARM array, when an alarm happen}
                VARs_TO_LOG[0].USINT := 0;                      (* Cleaning of "additional variable" *)
                VARs_TO_LOG[1].USINT := 0;

                CASE idx OF
                    1:  (*SAVING ADDITIONAL INFO (e.g.: Pressure/Temperature)*)
                        RFtrg_Alr1(CLK := Alarms.Arr[idx].Info.Trigger);

                        IF RFtrg_Alr1.Q THEN
                            VARs_TO_LOG[0].REAL := Prg_InputMng.Ain1Val;
                            VARs_TO_LOG[1].REAL := 99.99;
                        END_IF;

                    2:  (*SAVING ADDITIONAL INFO (e.g.: Error code/Temperature)*)
                        RFtrg_Alr2(CLK := Alarms.Arr[idx].Info.Trigger);

                        IF RFtrg_Alr2.Q THEN
                            VARs_TO_LOG[0].REAL := Prg_InputMng.Ain1Val;
                            VARs_TO_LOG[1].REAL := 99.99;
                        END_IF;
                    3:  (*SAVING ADDITIONAL INFO (e.g.: Pressure/Temperature)*)
                        RFtrg_Alr3(CLK := Alarms.Arr[idx].Info.Trigger);

                        IF RFtrg_Alr3.Q THEN
                            VARs_TO_LOG[0].REAL := Prg_InputMng.Ain1Val;
                            VARs_TO_LOG[1].REAL := 99.99;
                        END_IF;

                    4:  (*SAVING ADDITIONAL INFO (e.g.: Error code/Temperature)*)
                        RFtrg_Alr4(CLK := Alarms.Arr[idx].Info.Trigger);

                        IF RFtrg_Alr4.Q THEN
                            VARs_TO_LOG[0].REAL := Prg_InputMng.Ain1Val;
                            VARs_TO_LOG[1].REAL := 99.99;
                        END_IF;
                END_CASE;
            {ENDREGION}

            Alarms.Arr[idx]
                            (
                                DataVal         := VARs_TO_LOG, (* Remember to define ALARM_VALUES *)
                        	    AlrmRes         := AlrmRes,

                        	    Lst_ActAlrm     := Active_Alrm,
                        	    Lst_LogAlrm     := Log_Alarm,
                        	    Lst_LogAlrm_Idx := LogAlrmIdx
                            );
        END_FOR;
    {ENDREGION}

    {REGION CLEAN THE LOG ARRAY}
        IF LogAlrmRes THEN
            LogAlrmRes       := FALSE;
            (*RESTART LOG*)
            LogAlrmIdx := 0;

            (*CLEAR LOG LIST*)
            FOR idx := 1 TO TO_DINT(UPPER_BOUND(Log_Alarm, 1)) DO
                Log_Alarm[idx] := CleanLog;
            END_FOR;
        END_IF;
    {ENDREGION}

    {REGION GET ALARM CATEGORIES}
        ActAlr_ForCategory := Alarm_Mng(Active_Alrm);

                        //    := ActAlr_ForCategory.0;                       // BIT n.0  ->
        Al_SrsUnit            := ActAlr_ForCategory.1;                       // BIT n.1  -> CAT_AL_SRS_UNIT
        Al_SrsCirc1           := ActAlr_ForCategory.2 OR Al_SrsUnit;         // BIT n.2  -> CAT_AL_SRS_CIRC1
                        //    := ActAlr_ForCategory.3;                       // BIT n.3  ->
        Wrg_Regul             := ActAlr_ForCategory.4;                       // BIT n.4  -> CAT_WRG_REGUL
        Wrg_BoardMst          := ActAlr_ForCategory.5;                       // BIT n.5  -> CAT_WRG_BOARD_MST
                        //    := ActAlr_ForCategory.6;                       // BIT n.6  ->
        Wrg_Circ1             := ActAlr_ForCategory.7;                       // BIT n.7  -> CAT_WRG_CIRC1
                        //    := ActAlr_ForCategory.8;                       // BIT n.8  ->
                        //    := ActAlr_ForCategory.9;                       // BIT n.9  ->
        Wrg_HrsCounters       := ActAlr_ForCategory.10;                      // BIT n.10 -> CAT_WRG_HRSCOUNTER
                        //    := ActAlr_ForCategory.11;                      // BIT n.11 ->
                        //    := ActAlr_ForCategory.12;                      // BIT n.12 ->
                        //    := ActAlr_ForCategory.13;                      // BIT n.13 ->
                        //    := ActAlr_ForCategory.14;                      // BIT n.14 ->
        Al_Call_Service       := ActAlr_ForCategory.15;                      // BIT n.15 -> CAT_BLINK_KEY_SERVICE
    {ENDREGION}

    {REGION MANAGEMENT OF ALARM RELAY}
        (*Depending on alarm relay configuration, the alarm relay is activated by serious alarms only or by all alarms (including devices maintenance, retain memory,...) *)

        Al_RegulationAlrms :=    Al_SrsUnit
                              OR Al_SrsCirc1
                              OR Wrg_Regul;

        Al_MiscAlrms :=    Wrg_BoardMst
                        OR Wrg_Circ1
                        OR Wrg_HrsCounters;

        RelayAlrm := Al_RegulationAlrms OR (AlarmRelayCfg AND Al_MiscAlrms); // Dout RELAY
    {ENDREGION}

    {REGION COUNT OF TOTAL ALARMs AND WARNINGs ACTIVE}
        FOR idx := 1 TO TO_DINT(UPPER_BOUND(Active_Alrm,1)) DO
            IF Active_Alrm[idx] >= 1 THEN
                TotActAlm := TotActAlm + 1;
            END_IF;
        END_FOR;

        GblAlarm := UINT_TO_BOOL(TotActAlm);

        (*LED-ALARM and BUZZER*)
        IF TotActAlm > TotActAlm_Old THEN
            Req_FixLED_Alarm   := FALSE;    // LED-ALARM on
            Req_BlinkLED_Alarm := TRUE;     // LED-ALARM is blinking
            BuzzerSilenced     := FALSE;    // Buzzer is buzzing
        END_IF;

        TotActAlm_Old := TotActAlm;
    {ENDREGION}
END_PROGRAM

(* ---- 010_GENERAL_MNG.st ---- *)
USING System;
USING System.UI;
USING System.NFC;
USING System.Logs;
USING System.Text;
USING System.NVRAM;
USING System.Timer;
USING System.Serial;
USING System.Globalization;

USING Libs.GetTime_v0_1_8;
USING Libs.Blackout_v2_0_1;

VAR_GLOBAL
    (**Client is deleting memory*)
    ClientDeletingMem : BOOL;
END_VAR

PROGRAM Main
    VAR PUBLIC
    END_VAR
    VAR
        (**Client waiting time, before to delete memory*)
        TON_ClientWaitBefroreDelMem  : TON;
        (**FB Blackout*)
        Blackout1            : Blackout;
        (**Info saved in NVRAM*)
        NVRAM_Info : DWORD;
        (**This program calls other programs*)
        Prg_ProgramsExecutor : ProgramsExecutor;
        (**Save current system time *)
        {ATTRIBUTE UOM MILLISECOND}
        MemTime              : UDINT;
        (**First cycle*)
        FirstCycleDone       : BOOL;
        (**After restoring the memory to default, it waits 10s before restarting the PLC*)
        TON_WaitRestartPlc   : TON;
        (**R_TRIG Restore Default Settings*)
        Rtrg_RestoreDefault  : R_TRIG;
        (**Local time used to set RTC by network*)
        NewLocTimeByNet      : DateTime;
        (**Timezone POSIX string*)
        TzPOSIX              : STRING;
        (**Settings feedback of TimeZone *)
        Err_TimeZone         : UINT;
        (**Settings feedback of LocalTime*)
        Err_LocalTime        : UINT;
        (**Settings feedback of SetTime*)
        Err_SetTime          : UINT;
        i                    : DINT;
    END_VAR

    CurrSysT        := GetSystemTimeAdv();
    TaskMainCurrT   := GetTaskStartTimeAdv();
    TaskMainLiveCnt := GetTaskLiveCounter();
    RetainWrN       := TO_UDINT(GetRetainWritingsNumber());

    {REGION Read Date/Time}
        GetTime(TimeUTC);
        GetLocalTime(LocDateAndTime);
        GetLocalTime(LocTime);
        CurrLocTime.Hour        := LocTime.Hour;
        CurrLocTime.Minute      := LocTime.Minute;
        CurrLocTime.Second      := LocTime.Second;
        CurrLocTime.Millisecond := LocTime.Millisecond;
        CurrLocTime.Day         := LocTime.Day;
        CurrLocTime.Month       := LocTime.Month;
        CurrLocTime.Year        := LocTime.Year;
        Day_Week                := DAY_OF_WEEK(LocTime);
    {ENDREGION}

    {REGION First cycle}
        IF NOT FirstCycleDone THEN
            FirstCycleDone := TRUE;
            MemTime        := TaskMainCurrT;

            GetSystemInfo(SysInfo);
            GetHardwareDescription(HardwareInfo);
            GetModel(DeviceType, BoardType, MachineType, HwCode);
            GetProjectInfo(InfoProject);
            GetProductInfo(InfoProduct);
            GUID := SplitPrjGUID(InfoProject.ProjectID);

            (*The PLC is enabled to start only after checking the product code*)
            Go_PLC := TRUE;

            {REGION Balckout}
                (*Read*)
                NVRAM_ReadVar(0, NVRAM_Info);
                PwrOffDate_NVRAM_BLKO := TO_UDINT(NVRAM_Info);
            {ENDREGION}

            {REGION COMUNICATION IS STOPPED DURING INITIALIZATION OF INTERNAL PROTOCOLs STRUCTUREs.}
                (*BMS*)
//                Supervisor.Init(FALSE);
                (*Fieldbus*)
//                MBM_Line.Init(FALSE);
            {ENDREGION}

            {REGION IoT Third Parts Integration: Alarms retrieve via "Modbus File Transfer"}
               (*Following APIs calls are needed*)
                System.Alarm.AlarmInfoManagement(AlrmInfoArr);
                System.Alarm.AlarmLogManagement(LOG_ALARM);
            {ENDREGION}
        ELSE
            {REGION Balckout}
                (*Write*)
                NVRAM_Info := TO_DWORD(TO_UDINT(TimeUTC));
                NVRAM_WriteVar(0, NVRAM_Info);
                (*Read*)
                NVRAM_ReadVar(0, NVRAM_Info);
                PwrOffDate_NVRAM_BLKO :=  TO_UDINT(NVRAM_Info);
            {ENDREGION}
        END_IF;

        TaskMainExeT := TaskMainCurrT - MemTime;
        MemTime      := TaskMainCurrT;
    {ENDREGION}

    Blackout1(
                PwrOffDate_NVRAM   := PwrOffDate_NVRAM_BLKO,

                OffMins            => OffMins_BLKO,
                OffHours           => OffHours_BLKO,
                OffDays            => OffDays_BLKO,

                LastOnSec          => LastOnSec_BLKO,
                LastOnMin          => LastOnMin_BLKO,
                LastOnHour         => LastOnHour_BLKO,
                LastOnDay          => LastOnDay_BLKO,
                LastOnMonth        => LastOnMonth_BLKO,
                LastOnYear         => LastOnYear_BLKO
                );

    {REGION RESTORE PLC MEMORY TO DEFAULT SETTINGS}
        Rtrg_RestoreDefault(CLK := RestoreDefault);

        IF Rtrg_RestoreDefault.Q THEN           (*Saving BMS2 settings before restoring memory*)
            BMS2_Addr_SavedRAM := BMS2_Addr;
            BMS2_Baud_SavedRAM := BMS2_Baud;
            BMS2_Conf_SavedRAM := BMS2_Conf;
        END_IF;

        TON_ClientWaitBefroreDelMem(IN := RestoreDefault AND NOT ClientDeletingMem, PT := T#5s); (*NOTE: In a net "CLIENT + SERVER": server must receive the restore memory command -> then after a delay -> client can restore its memory*)

        IF TON_ClientWaitBefroreDelMem.Q THEN
            ClientDeletingMem := TRUE;
            RetainRestoreDefault();             (*NOTE: This request will be executed at END of MAIN task.*)
        END_IF;
    {ENDREGION}

    {REGION DATE AND TIME}
        {REGION SETTINGS pCO CLOCK TIME BY APPLICA}
            IF APPsCfgRTC.SetRTC THEN
                APPsCfgRTC.SetRTC := FALSE;
                //Necessary and in this order
                Err_TimeZone := SetTimeZone(APPsCfgRTC.TimeZone);
                Err_SetTime  := SetTime(APPsCfgRTC.DateTime);           (*APPLICA give UTC Time*)

                {REGION Saving of time ZONE when RTC set by APPs}
                    FOR i := LOWER_BOUND(TimeZonePOSIX, 1) TO UPPER_BOUND(TimeZonePOSIX, 1) DO
                        IF APPsCfgRTC.TimeZone = TimeZonePOSIX[i] THEN
                            Timezone := TO_UINT(i);
                            EXIT;
                        END_IF;
                    END_FOR;
                {ENDREGION}
            END_IF
        {ENDREGION};

        {REGION SETTINGS pCO CLOCK TIME BY USER NETWORK}
            IF SetClockByNet THEN
                SetClockByNet := FALSE;

                NewLocTimeByNet.Day    := NewDateTimeByNet.Day;                 (*NOTE: Necessary to adjust TYPE to UINT*)
                NewLocTimeByNet.Month  := NewDateTimeByNet.Month;
                NewLocTimeByNet.Year   := NewDateTimeByNet.Year;

                NewLocTimeByNet.Hour   := NewDateTimeByNet.Hour;
                NewLocTimeByNet.Minute := NewDateTimeByNet.Minute;
                NewLocTimeByNet.Second := NewDateTimeByNet.Second;

                TzPOSIX := TimeZoneName[Timezone];
                //Necessary and in this order
                Err_TimeZone  := SetTimeZone(TzPOSIX);                          // WAIT API by OS!
                Err_LocalTime := SetLocalTime(NewLocTimeByNet);
            END_IF;
        {ENDREGION}
    {ENDREGION}

    {REGION BMS/FIELDBUS SERIAL PORTs CONFIGURATION}
//        CASE UoMZoneHMI OF
//            UOM_ZONE#SI:
//                Supervisor.Info.Zone := SI;
//                // Server BMS uses only SI to communicate (Client FielBus <-> Server BMS)
//                // NOTE: In a net CLIENT+SERVER set NoConverion =0 beetwen: Client FielBus <-> Server BMS to increase pCO speed
//                // i.e.: FBnet.Info.Zone=0 and BMSnet.Info.Zone=0
//            UOM_ZONE#Imperial:
//                Supervisor.Info.Zone := Imperial;
//        ELSE
//            Supervisor.Info.Zone := NONE;
//        END_CASE;

        {REGION CHANGE BMS2 SETTINGS}
            {REGION PROCEDURE TO RESTORE BMS2 SETTINGS}
                (*Memory after deleting command is immediately ready the next cycles*)
                IF ClientDeletingMem THEN
                    // Restore BMS2 settings
                    BMS2_Addr := BMS2_Addr_SavedRAM;
                    BMS2_Baud := BMS2_Baud_SavedRAM;
                    BMS2_Conf := BMS2_Conf_SavedRAM;

                    // Force update BMS2 settings
                    Bms2_ChangeSet := TRUE;
                END_IF;
            {ENDREGION}

            IF Bms2_ChangeSet THEN
                Bms2_ChangeSet := FALSE;
//                  SetupSerialSettings(Line_cPCOe2.SerialSettings, BMS2_Baud, BMS2_Conf);
//                SetupSerialSettings(Supervisor.SerialSettings, BMS2_Baud, BMS2_Conf);

                // Change BMS address
//                Supervisor.ChangeIdent(BMS2_Addr);

                // Change setting of BMS supervisor port
//                Supervisor.ChangeSettings();

                // Set the same settings for BMS port on Default app (NOTE: In case of FW ugrade the device will be reachable with the previous settings)
//                SaveIdePortSettings(Supervisor.SerialSettings.Channel, Supervisor.SerialSettings.Speed, Supervisor.SerialSettings.Bits, Supervisor.SerialSettings.Parity, Supervisor.SerialSettings.Stops, BMS1_Addr);
            END_IF;

//            BMS2_Online := Supervisor.Info.Online OR Dbg_BMS2Online;
        {ENDREGION}

        {REGION CHANGE FIELDBUS2 SETTINGS}
//            IF FB2_ChangeSet THEN
//                FB2_ChangeSet := FALSE;

//                SetupSerialSettings(MBM_Line.SerialSettings, FB2_Baud, FB2_Conf);

//                // Change setting of FB supervisor port
//                MBM_Line.ChangeSettings();
//            END_IF;
        {ENDREGION}
    {ENDREGION}

    {REGION READ BUFFER OF EACH SERIAL PORT}
        // NOTE: when the protocols are in START the read() method obtain the variables
        //       from each buffer -> so the variables can be used inside STone.

        // BMS
//        Supervisor.Read();
        // Fieldbus
//        MBM_Line.Read();
    {ENDREGION}

    //------ CALL OF PROGRAMs ---------
    IF NOT ClientDeletingMem THEN
        Prg_ProgramsExecutor();
    END_IF;
    //---------------------------------

    {REGION WRITE BUFFER OF EACH SERIAL PORT}
        IF ClientDeletingMem THEN
            //Stop all protocols.
//            Supervisor.Stop();
//            MBM_Line.Stop();
        ELSE
            {REGION BMS: WRITE VARIABLES}
                //Modbus Server line
//                Supervisor.Write();
                //START COMMUNICATION
//                Supervisor.Start();
            {ENDREGION}

            {REGION FIELDBUS: WRITE VARIABLES}
                //Modbus Client line
//                MBM_Line.Write();
                //START COMMUNICATION
//                MBM_Line.Start();
            {ENDREGION}
        END_IF;
    {ENDREGION}

	(* Refresh UI *)
	SendVirtualKey(NO_KEY, 1);

    //------------------------------------------------------------------------------------
    //------------ WARM SOFTWARE RESET----------------------------------------------------
    //------------------------------------------------------------------------------------
    TON_WaitRestartPlc(IN := ClientDeletingMem, PT := T#6s);
    IF TON_WaitRestartPlc.Q THEN
        // Wait 6s because Retain will be write every 5s
        // 0 - WARM start;
        SoftwareReset(0);
    END_IF;
END_PROGRAM

(* ---- 015_ProgramsExecutor.st ---- *)
USING System;
USING System.Text;
USING System.Timer;

VAR_GLOBAL
    {REGION INSTANCES OF PROGRAMs}
        Prg_NetFieldbus_Read  : NetFieldbus_Read;
//      Prg_Unitconfig        : Unitconfig;
        Prg_InputMng          : InputMng;
        Prg_AlarmsMng         : AlarmsMng;
        Prg_StoreAlarms       : StoreAlarms;
        Prg_OnOffUnit         : OnOffUnit;
//      Prg_Regulation        : Regulation;
        Prg_HoursCounterMng   : HoursCounterMng;
        Prg_OutputMng         : OutputMng;
        Prg_NetFieldbus_Write : NetFieldbus_Write;
        Prg_uPC2EMCMain       : uPC2EMCMain;
    {ENDREGION}

    (**Delay of activation programs execution*)
    TON_StartExcPrgs          : TON;

    SwSafeUpload              : SoftwareSafeUpload;
END_VAR

(*
  Insert here all the programs to be executed in your strategy.
 *)
PROGRAM ProgramsExecutor
    SwSafeUpload(KeybOffOn := KeybOnOff, StartUpload := NOT KeybOnOff);

    (*Read Fieldbus netwok*)
    Prg_NetFieldbus_Read();

    //Prg_Unitconfig();
    //Prg_InputMng();

    TON_StartExcPrgs(IN := Go_PLC, PT := T#10s);

    IF TON_StartExcPrgs.Q THEN
        Prg_AlarmsMng();
        Prg_StoreAlarms();
        //Prg_InputMng();
        //Prg_OnOffUnit();
        //Prg_Regulation();

        //Prg_HoursCounterMng();
        //Prg_Chiller();
        Prg_uPC2EMCMain();
        //Prg_OutputMng();

        (*Log management*)
        //Logs.Check();
    ELSE
        (*During pCO start up the display shows OFF*)
        UnitOff := TRUE;
    END_IF;

    (*Write Fieldbus netwok*)
    Prg_NetFieldbus_Write();
END_PROGRAM

(* ---- 020_NetFieldub_Read.st ---- *)
USING System;
USING System.Timer;

VAR_GLOBAL
    Dly_EnTmplate: TON;
END_VAR

PROGRAM NetFieldbus_Read

        //==============================================
        // ENABLING OF TEMPLATE
        //==============================================
//        ClientModbus_pCO.Info.Enabled := En_FB1;

        //==============================================
        // READ FROM TEMPLATE IF SERVER IS ONLINE
        //==============================================
//        Dly_EnTmplate(IN := ClientModbus_pCO.Info.Enabled, PT := T#3s);
        //# Alarms.Table.Al_ServerOffline.Info.Trigger := Dly_EnTmplate.Q  AND (NOT ClientModbus_pCO.Info.IsOnline);

        //==============================================
        // COMUNICATION BETWEEN CLIENT/SALVE BAORD
        //==============================================
    	IF En_FB1 THEN

            {REGION READS FROM SERVER BOARD (INPUT STATUS -> COILS)}

                //..........................................
                // PUT HERE YOUR VARIABLEs
                //..........................................
            // := ClientModbus_pCO.IR_0_CANCELLAMI5;
            {ENDREGION}

            {REGION READS PARAMETERS FROM SERVER BOARD (INPUT REGISTER)}
                //# RemProbeT := ClientModbus_pCO.IR_00_RemProbeT;

                //..........................................
                // PUT HERE YOUR VARIABLEs
                //..........................................
            // := ClientModbus_pCO.IS_0_CANCELLAMI6;
            {ENDREGION}
    END_IF;

END_PROGRAM

(* ---- 030_InputMng.st ---- *)
USING System;
USING System.IO;

USING Libs.AinMng_v2_0_1;

VAR_GLOBAL PERSISTENT
    (**Offeset of Ain1 probe*) {METADATA MIN_VAL -99.9}  {METADATA MAX_VAL 99.9}
    Ain1PrbOffset: REAL;
    (**Din1 relè logic. Logic to manage an ALARM (FALSE=NC, TRUE=NO).*)
    Din1Logic : BOOL := DIN_LOGIC_NC;
    (**Din2 relè logic. Logic to manage a COMMAND (FALSE=NC, TRUE=NO).*)
    Din2Logic : BOOL := DIN_LOGIC_NO;
END_VAR

PROGRAM InputMng
    VAR PUBLIC
        (**Din1 value (used as Remote unit alarm)*)
        Din1    : BOOL;
        (**Din2 value (used as Remote OnOff unit)*)
        Din2    : BOOL;
        (**Ain1 value*) {ATTRIBUTE UOM CELSIUS} {METADATA MIN_VAL -99.9} {METADATA MAX_VAL 99.9}
        Ain1Val : REAL;
    END_VAR
    VAR
        (**AinMng function block*)
        Ain1  : AinMng;
    END_VAR

    {REGION Din1: Unit remote alarm}
        Din1 := ID[1] XOR Din1Logic;
    {ENDREGION}

    {REGION Din2: Unit ON/OFF command}
        Din2 := ID[2] XOR Din2Logic;
    {ENDREGION}

    {REGION Ain1: NTC probe}
        uConfig[1].mode_sel  := LIB_IO_AIN;                 (*Configuration of Ain1 as AIN*)
        uConfig[1].mode_type := LIB_IO_PROBE_NTC;           (*Configuration of Ain1 probe as NTC*)
        uConfig[1].filter    := PRB_FILTER;

        Ain1(
                Ain       := U[1].r,
                AinType   := uConfig[1].mode_sel,
                PrbOffset := Ain1PrbOffset,
              //MinVal    := REAL,
              //MaxVal    := REAL,
                AlrmDT    := PrbDly,

                En_FB     := TRUE,

                PrbVal    => Ain1Val
              //OnOffVal  => BOOL
              //PrbAlrm   =>...
            );
        Alarms.Table.Al_Ain1Alrm.Info.Trigger := Ain1.PrbAlrm; // NOTE: is possible check -> (uConfig[1].error <> LIB_IO_NO_ERR)
    {ENDREGION}

END_PROGRAM

(* ---- 040_AlarmsMng.st ---- *)
USING System;
USING System.Math;
USING System.Timer;
VAR_GLOBAL
    EEpRetainErrorOccurred : BOOL := FALSE;
    event : Event;
    error : DINT;
    taskId : INT;
    Err_ID : INT(0..100);
END_VAR

{DEFINE Diff_ALM_U_NTC  0.5}
{DEFINE Diff_ALM_U_V  0.3}
{DEFINE Diff_ALM_U_A  0.36}

PROGRAM AlarmsMng

    VAR_TEMP
        i : INT;
    END_VAR

    {REGION ExceptionInstance}
        Alarms.Table.Al_RetainSavedTooOften.Info.Trigger := ExceptionInstance.ExceptionError = ERR_RETAIN_SAVE_TOO_OFTEN;
        Alarms.Table.Al_NFCSavedTooOften.Info.Trigger    := ExceptionInstance.ExceptionError = ERR_NFC_SAVE_TOO_OFTEN;
        ExceptionInstance.ExceptionError                 := 0;   (*PAY ATTENTION! Reset of output.*)
    {ENDREGION}
    GetCurrentEvent(event);
    IF event.EventType = VMSystemEvent AND event.Mask = TO_DWORD(EVENT_EXCEPTION) THEN
        taskId := TO_INT(event.Data);
        GetLastTaskErrorCodeError(taskId, error);
        CASE error OF
            ERR_RETAIN_INIT_FAIL,
            ERR_RETAIN_NOT_INTITIALIZED,
            ERR_RETAIN_BEGIN_FAIL,
            ERR_RETAIN_WRITE_BLOCK_FAIL,
            ERR_RETAIN_END_FAIL,
            ERR_RETAIN_BACKUP_FAIL,
            ERR_RETAIN_READ_BLOCK_FAIL,
            ERR_RETAIN_CORRUPTED,
            ERR_RETAIN_ERROR_ACCESS,
            ERR_RETAIN_WRITING_ERROR,
            ERR_RETAIN_READING_ERROR:
                EEpRetainErrorOccurred := TRUE;
        END_CASE;
        (*Resume the task, reset the task error*)
        ResumeTask(taskId, error, 0);
    END_IF;

//    Alarms.Table.Al_Din1Alrm.Info.Trigger := Prg_InputMng.Din1 AND En_DinAlrm;

//    //High Temperature alarms
//    IF W_InTemp>=15.0 AND Unit_On_Off THEN
//        Alarms.Table.Al_HiTemp.Info.Trigger := TRUE;
//    ELSE
//        Alarms.Table.Al_HiTemp.Info.Trigger := FALSE;
//    END_IF;

//    //Antifreese alaem
//    Alarms.Table.Al_Afreese.Info.Trigger := W_InTemp<=3.0 AND Unit_On_Off;

//    //Broken probe alarm
//    Alarms.Table.Al_Prb.Info.Trigger := AL_Prb_W_InTemp;
    FOR i := 1 TO 24 DO
        CASE i OF
            1, 2, 4, 5, 7, 10, 11, 12, 14:
                InputValAlarms[i] := InputValueR[i] > 7.5+Diff_ALM_U_NTC OR InputValueR[i] < 7.5-Diff_ALM_U_NTC;
            3:
                InputValAlarms[i] := InputValueR[i] > 2.5+Diff_ALM_U_V OR InputValueR[i] < 2.5-Diff_ALM_U_V;
            6:
                InputValAlarms[i] := InputValueR[i] > 1.0+Diff_ALM_U_V OR InputValueR[i] < 1.0-Diff_ALM_U_V;
            8,13:
                InputValAlarms[i] := InputValueR[i] > 5.0+Diff_ALM_U_V OR InputValueR[i] < 5.0-Diff_ALM_U_V;
            9:
                InputValAlarms[i] := InputValueR[i] > 12.0+Diff_ALM_U_A OR InputValueR[i] < 12.0-Diff_ALM_U_A;

            ELSE
                InputValAlarms[i] :=(DInputValue[i - 14] XOR DefaultDInputValue[i - 14]);
        END_CASE;
    END_FOR;

    Err_ID := 0;
    FOR i := 1 TO TO_INT(noAlrms) DO
        IF Active_Alrm[i]<>0 THEN
            Err_ID := i;
            EXIT;
        END_IF;
    END_FOR;
        Alarms.Table.Al_U1_PrbAlrm.Info.Trigger := AinAlarms[1];
        Alarms.Table.Al_U2_PrbAlrm.Info.Trigger := AinAlarms[2];
        Alarms.Table.Al_U3_PrbAlrm.Info.Trigger := AinAlarms[3];
        Alarms.Table.Al_U4_PrbAlrm.Info.Trigger := AinAlarms[4];
        Alarms.Table.Al_U5_PrbAlrm.Info.Trigger := AinAlarms[5];
        Alarms.Table.Al_U6_PrbAlrm.Info.Trigger := AinAlarms[6];
        Alarms.Table.Al_U7_PrbAlrm.Info.Trigger := AinAlarms[7];
        Alarms.Table.Al_U8_PrbAlrm.Info.Trigger := AinAlarms[8];
        Alarms.Table.Al_U9_PrbAlrm.Info.Trigger := AinAlarms[9];
        Alarms.Table.Al_U10_PrbAlrm.Info.Trigger := AinAlarms[10];
        Alarms.Table.Al_U11_PrbAlrm.Info.Trigger := CurrentIOInfo.U>10 AND AinAlarms[11];
        Alarms.Table.Al_U12_PrbAlrm.Info.Trigger := CurrentIOInfo.U>11 AND AinAlarms[12];
        Alarms.Table.Al_U1_ValAlrm.Info.Trigger := InputValAlarms[1];
        Alarms.Table.Al_U2_ValAlrm.Info.Trigger := InputValAlarms[2];
        Alarms.Table.Al_U3_ValAlrm.Info.Trigger := InputValAlarms[3];
        Alarms.Table.Al_U4_ValAlrm.Info.Trigger := InputValAlarms[4];
        Alarms.Table.Al_U5_ValAlrm.Info.Trigger := InputValAlarms[5];
        Alarms.Table.Al_U6_ValAlrm.Info.Trigger := InputValAlarms[6];
        Alarms.Table.Al_U7_ValAlrm.Info.Trigger := InputValAlarms[7];
        Alarms.Table.Al_U8_ValAlrm.Info.Trigger := InputValAlarms[8];
        Alarms.Table.Al_U9_ValAlrm.Info.Trigger := InputValAlarms[9];
        Alarms.Table.Al_U10_ValAlrm.Info.Trigger := InputValAlarms[10];
        Alarms.Table.Al_U11_ValAlrm.Info.Trigger := CurrentIOInfo.U>10 AND InputValAlarms[11];
        Alarms.Table.Al_U12_ValAlrm.Info.Trigger := CurrentIOInfo.U>11 AND InputValAlarms[12];
        Alarms.Table.Al_DI1Alrm.Info.Trigger := InputValAlarms[15];
        Alarms.Table.Al_DI2Alrm.Info.Trigger := InputValAlarms[16];
        Alarms.Table.Al_DI3Alrm.Info.Trigger := InputValAlarms[17];
        Alarms.Table.Al_DI4Alrm.Info.Trigger := InputValAlarms[18];
        Alarms.Table.Al_DI5Alrm.Info.Trigger := EVD_EVOinstance.DeviceEvdEvo.Info.isOnline AND InputValAlarms[19];
        Alarms.Table.Al_DI6Alrm.Info.Trigger := EVD_EVOinstance.DeviceEvdEvo.Info.isOnline AND InputValAlarms[20];
        Alarms.Table.Al_DI7Alrm.Info.Trigger := CurrentIOInfo.ID > 6 AND InputValAlarms[21];
        Alarms.Table.Al_DI8Alrm.Info.Trigger := CurrentIOInfo.ID > 7 AND InputValAlarms[22];
        Alarms.Table.Al_DI9Alrm.Info.Trigger := CurrentIOInfo.ID > 8 AND InputValAlarms[23];
        Alarms.Table.Al_DI10Alrm.Info.Trigger := CurrentIOInfo.ID > 9 AND InputValAlarms[24];
        Alarms.Table.Al_cPCOe1ERR.Info.Trigger := Cpcoe1_Err;
        Alarms.Table.Al_cPCOe2ERR.Info.Trigger := Cpcoe2_Err;
        Alarms.Table.Al_cPCOe3ERR.Info.Trigger := CurrentIOInfo.NO > 10 AND Cpcoe3_Err;
        Alarms.Table.Al_DisplayERR.Info.Trigger :=NOT DisplayIsOnline;
        Alarms.Table.Al_BMS1ERR.Info.Trigger :=NOT pCOWeb_BMS1.Info.Online;
        Alarms.Table.Al_ETH1ERR.Info.Trigger :=NOT Supervisor_ETH1.Info.Online;
        Alarms.Table.Al_ValveDriveERR.Info.Trigger:= EVD_EVOinstance.DeviceEvdEvo.Info.isOnline AND (EVD_EVO_MBSErr.DevErr<>0 OR EVD_EVO_Alr.Al_ConnectionBoardDrvB OR EVD_EVO_Alr.Al_EEPROM OR EVD_EVO_Alr.Al_EmergencyClosing
                                                                                                    OR EVD_EVO_Alr.Al_HwIncompatible OR EVD_EVO_Alr.Al_IncompleteClosing OR EVD_EVO_Alr.Al_MotorVlvA OR EVD_EVO_Alr.Al_MotorVlvB);
        Alarms.Table.Al_S1_Alrm.Info.Trigger := EVD_EVOinstance.DeviceEvdEvo.Info.isOnline AND (EVD_EVO_S1Value > 5.3 OR EVD_EVO_S1Value < 4.7 OR EVD_EVO_S1Alarm);
        Alarms.Table.Al_S2_Alrm.Info.Trigger := EVD_EVOinstance.DeviceEvdEvo.Info.isOnline AND (EVD_EVO_S2Value > 8.0 OR EVD_EVO_S2Value < 7.0 OR EVD_EVO_S2Alarm);
        Alarms.Table.Al_S3_Alrm.Info.Trigger := EVD_EVOinstance.DeviceEvdEvo.Info.isOnline AND (EVD_EVO_S3Value > 5.3 OR EVD_EVO_S3Value < 4.7 OR EVD_EVO_S3Alarm);
        Alarms.Table.Al_S4_Alrm.Info.Trigger := EVD_EVOinstance.DeviceEvdEvo.Info.isOnline AND (EVD_EVO_S4Value > 8.0 OR EVD_EVO_S4Value < 7.0 OR EVD_EVO_S4Alarm);
END_PROGRAM

(* ---- 060_OnOffUnit.st ---- *)
USING system;
USING System.Math;
USING System.Timer;

PROGRAM OnOffUnit

    {REGION UNIT ON/OFF COMMAND}
        UnitOn :=       NOT Al_SrsUnit
                    AND KeybOnOff
                    AND (NOT En_DinAlrm OR NOT Prg_InputMng.Din1)                   (* Remote Alarm*)
                    AND (NOT En_DinOffOn OR Prg_InputMng.Din2)                      (**)
                    AND (NOT (En_BmsOffOn AND BMS2_Online) OR BmsOffOn);            (*Unit works in stand-alone mode in case of BMS offline!*)

        UnitOff := NOT UnitOn;

        (*UNIT STATUS*)
        IF En_DinOffOn AND NOT Prg_InputMng.Din2 THEN
            UnitStatus := UNIT_STATUS#OffByDI;
        ELSIF  NOT KeybOnOff THEN
            UnitStatus := UNIT_STATUS#OffByKeyboard;
        ELSIF En_BmsOffOn AND BMS2_Online AND NOT BmsOffOn THEN
            UnitStatus := UNIT_STATUS#OffByBMS;
        ELSIF Al_SrsUnit THEN
            UnitStatus := UNIT_STATUS#OffByAlarm;
        ELSIF UnitOn THEN
            UnitStatus := UNIT_STATUS#UnitON;
        END_IF;
    {ENDREGION}

END_PROGRAM

(* ---- 070_HoursCounterMng.st ---- *)
USING System;
USING System.Math;
USING System.Timer;

USING Libs.Counters;

PROGRAM HoursCounterMng
    VAR
        (**Unit On HoursCounter FB*)
        HrsCntr_UnitOn : HoursCounter;
        (**Used for debug: n° of seconds for hour (Set 0=3600s)*)
        HrsCntrAdjust  : UINT;

    END_VAR

    {REGION UNIT}
        HrsCntr_UnitOn(
                        In             := UnitOn,
                        ThrshAlrm      := 50*100,                       (* Threshold in hundreds *)
                        HrsPrstUpdRate := HRS_PRST_UPD_RATE,
                        Adjust         := HrsCntrAdjust,
                        ResAlrm        := UnitOnResHrs,
                        ResTotCnt      := ResTotCnt,

                        Hours          => UnitOnHrs,
                      //Alrm           => BOOL,                         (* PAY ATTENTION! Connect here your alarm *)

                        Partial_PRST   := UnitOnHrsPartial,
                        Total_PRST     := UnitOnHrsTot
                    );

        IF UnitOnResHrs THEN
            UnitOnResHrs := FALSE;                                      (* Auto-Reset *)
        END_IF;
    {ENDREGION}

    (*--------------------------------
               HOURS COUNTER RESET
      --------------------------------*)
    IF ResTotCnt THEN
        ResTotCnt := FALSE;                                             (* Auto-Reset *)
    END_IF;
END_PROGRAM
